(* Timer activ *)
	TimerOn(IN:=TRUE,PT:=T_Cylinder.T_Config.tDelayOn);
	TimerOff(IN:=TRUE,PT:=T_Cylinder.T_Config.tDelayOff);
	TimerPreOn(IN:=TRUE,PT:=T_Cylinder.T_Config.tDelayPreOn);
	TimerPreOff(IN:=TRUE,PT:=T_Cylinder.T_Config.tDelayPreOff);
	TimerOut(IN:=TRUE,PT:=T_Cylinder.T_Config.tTimeOut);
	TimerActiv(IN:=TRUE,PT:=T_Cylinder.T_CtrleCyl.T_Standard.tDelayActiv);
	TimerAfterSensorOn(IN:=TRUE,PT:=T_Cylinder.T_CtrleCyl.T_Standard.tDelayAfterSensorOn);
	TimerAfterSensorOff(IN:=TRUE,PT:=T_Cylinder.T_CtrleCyl.T_Standard.tDelayAfterSensorOff);
(* waiting for activ *)
	IF NOT(T_Cylinder.T_CtrleCyl.xErr) THEN
		CASE iStep OF
		(* process timer On *)
		1:	IF (T_Cylinder.T_Config.tDelayPreOn = T#0s) THEN
				TimerOn(IN:=FALSE);
				xCylinder:=T_Cylinder.T_Config.xActivState;
				T_Cylinder.T_CtrleCyl.T_Standard.xActivOn:=TRUE;
				iStep:=2;
			ELSE
				TimerPreOn(IN:=FALSE);
				iStep:=4;
			END_IF;
		(* wait for timer On *)
		2:	IF TimerOn.Q THEN
				iStep:=3;
				TimerOut(IN:=FALSE);
			END_IF
		(* control position activ *)
		3:	IF T_Cylinder.T_Config.xCtrlePosOn THEN
			(* position ctrle activ *)
				IF TimerOut.Q THEN
				(* timerout done, activ error cylinder has not activ position reached *)
					iStep:=999;
				ELSE
					IF xCtrlePosOn THEN
					(* Activ position reached, activ confirmation *)
						iStep:=80;
					END_IF
				END_IF
			ELSE
			(* no position ctrle, activ confirm *)
				iStep:=90;
			END_IF
		(* wait for timer Pre On *)
		4:	IF TimerPreOn.Q THEN
				T_Cylinder.T_Config.tDelayPreOn:=T#0s;
				iStep:=1;
			END_IF
		(* process timer Off *)
		11:	IF (T_Cylinder.T_Config.tDelayPreOff = T#0s) THEN
				TimerOff(IN:=FALSE);
				xCylinder:=NOT(T_Cylinder.T_Config.xActivState);
				T_Cylinder.T_CtrleCyl.T_Standard.xActivOn:=FALSE;
				iStep:=12;
			ELSE
				TimerPreOff(IN:=FALSE);
				iStep:=14;
			END_IF;
		(* wait for timer Off *)
		12:	IF TimerOff.Q THEN
				iStep:=13;
				TimerOut(IN:=FALSE);
			END_IF
		(* control position inactiv *)
		13:	IF T_Cylinder.T_Config.xCtrlePosOff THEN
			(* control position activ *)
				IF TimerOut.Q THEN
				(* timerout done, activ error 'cylinder has not inactiv position reached' *)
					iStep:=998;
				ELSE
					IF xCtrlePosOff THEN
					(* inactiv position reached, activ confirmation *)
						iStep:=85;
					END_IF
				END_IF
			ELSE
			(* no control position activ, activ confirmation *)
				iStep:=99;
			END_IF
		(* wait for timer Pre Off *)
		14:	IF TimerPreOff.Q THEN
				T_Cylinder.T_Config.tDelayPreOff:=T#0s;
				iStep:=11;
			END_IF
		(* inverse cylinder state *)
		51:	xCylinder:=NOT(xCylinder);
			T_Cylinder.T_CtrleCyl.T_Standard.xActivOn:=NOT(T_Cylinder.T_CtrleCyl.T_Standard.xActivOn);
			iStep:=99;
		80:	IF (T_Cylinder.T_CtrleCyl.T_Standard.tDelayAfterSensorOn <> T#0s) THEN
				TimerAfterSensorOn(IN:=FALSE);
				iStep:=81;
			ELSE
				iStep:=90;
			END_IF;
		(* wait for time after sensor *)
		81:	IF TimerAfterSensorOn.Q THEN
				iStep:=90;
			END_IF
		85:	IF (T_Cylinder.T_CtrleCyl.T_Standard.tDelayAfterSensorOff <> T#0s) THEN
				TimerAfterSensorOff(IN:=FALSE);
				iStep:=86;
			ELSE
				iStep:=99;
			END_IF;
		(* wait for time after sensor *)
		86:	IF TimerAfterSensorOff.Q THEN
				iStep:=99;
			END_IF
		(* test if delay activ *)
		90:	IF T_Cylinder.T_CtrleCyl.T_Standard.tDelayActiv <> T#0s THEN
				TimerActiv(IN:=FALSE);
				iStep:=98;
			ELSE
				iStep:=99;
			END_IF
		(* wait for time delay activ *)
		98:	IF TimerActiv.Q THEN
			(* activ time is over, set variable off *)
				xCylinder:=NOT(T_Cylinder.T_Config.xActivState);
				T_Cylinder.T_CtrleCyl.T_Standard.xActivOn:=FALSE;
				iStep:=99;
			END_IF
		(* process end *)
		99:	T_Cylinder.T_CtrleCyl.xDone:=TRUE;
			T_Cylinder.T_CtrleCyl.xErr:=FALSE;
			T_Cylinder.T_CtrleCyl.udiErrorID:=16#0;
		(* error, cylinder not in inactiv position *)
		998:	T_Cylinder.T_CtrleCyl.xDone:=FALSE;
			T_Cylinder.T_CtrleCyl.xErr:=TRUE;
			T_Cylinder.T_CtrleCyl.udiErrorID:=16#F202;
		(* error, cylinder not in activ position *)
		999:	T_Cylinder.T_CtrleCyl.xDone:=FALSE;
			T_Cylinder.T_CtrleCyl.xErr:=TRUE;
			T_Cylinder.T_CtrleCyl.udiErrorID:=16#F201;
		END_CASE
	END_IF;
END_FUNCTION_BLOCK

(* POU GENERAL/FB_CalcSpindleForce, ST *)
FUNCTION_BLOCK FB_CalcSpindleForce
VAR_INPUT
	rForcePistonIn:REAL;	(* in Newton *)
	rPistonDiameterD1:REAL;	(* in mm *)
	rPistonDiameterD2:REAL;	(* in mm *)
	rMaxAirpressure:REAL;		(* in bar *)
	rMaxServoVoltage:REAL;	(* in Volt *)
END_VAR
VAR_OUTPUT
	iAnalogOutput:INT;		(* range 0 - 32767 *)
	rSetMaxForce:REAL;		(* in Newton *)
	rForcePistonOut:REAL;	(* in Newton *)
END_VAR
VAR
	rMaxForce: REAL;
	rAreaOutside: REAL;
	rArea: REAL;
	rTmpMaxAirpressure: REAL;
	rTmpAnalogOut:REAL;
	rMaxDigitAnalogOutput: REAL;
END_VAR
	rMaxDigitAnalogOutput:=(32767.0 / 10.0) * rMaxServoVoltage;
	rAreaOutside:=((rPistonDiameterD1/2.0)*(rPistonDiameterD1/2.0))*PI;
	rArea:=ABS(rAreaOutside) * 2.0;	(* the new spindle has two piston *)
	rArea:=rArea / 1000000.0;	(* Umwandeln von mm^2 in m^2 *)
	rTmpMaxAirpressure:=rMaxAirpressure * 100000.0;	(* convert from bar to pascal *)
	rMaxForce:=rArea * rTmpMaxAirpressure;
	rSetMaxForce:=rMaxForce;
	IF(rMaxForce = 0) THEN rMaxForce:=0.01; END_IF;	(* check divide by zero *)
	IF(rMaxForce <> 0.0) THEN
		rTmpAnalogOut:=(rForcePistonIn/rMaxForce)*rMaxDigitAnalogOutput;
		IF (rTmpAnalogOut > rMaxDigitAnalogOutput) THEN
			iAnalogOutput:=REAL_TO_INT(rMaxDigitAnalogOutput);
		ELSE
			iAnalogOutput:=REAL_TO_INT(rTmpAnalogOut);
		END_IF;
		rForcePistonOut:=rForcePistonIn;
	ELSE
		iAnalogOutput:=0;
		rForcePistonOut:=0;
	END_IF;
END_FUNCTION_BLOCK

(* POU GENERAL/FB_TorqueLevelAirPressureAnalog, ST *)
FUNCTION_BLOCK FB_TorqueLevelAirPressureAnalog
VAR_INPUT
	xActiveWorkProcess:BOOL;
	xBlockOutput:BOOL;
	rForceIn:REAL;			(* Range 0 - MaxTorque (mNm) *)
	T_Station_Parameter:ST_RETAIN_DATA_STATIONWORK;
	lrZ1ActualPosition:LREAL;
	xCylHCActive:BOOL;
END_VAR
VAR_OUTPUT
	iAnalogOutput:INT;		(* Range 0 - 32767 *)
	rForceOut:REAL;			(* Range 0 - MaxTorque (mNm) *)
	rMaxTorque:REAL;		(* mNm *)
END_VAR
VAR_IN_OUT
	TCylTorque:ST_CYLINDER;
END_VAR
VAR
	rTorque:REAL;
	rTorqueEndPosition:REAL;
	rAirPressureP:REAL;
	rDiffTorqueLEvel:REAL;
(* Tmp variable *)
	rMaxAirPressure: REAL;
	rTmpAnalogOut:REAL;
	rTmpForceOut: REAL;
	rPistonArea: REAL;
	rGearRatioGearBox: REAL;
	rPlanetCarrier: REAL;
	rGearRatioRocker: REAL;
	rMaxTmpAirPressure: REAL;
	rTorqueStartPosition: REAL;
	rZ1Position: REAL;
	rZ1Length: REAL;
	rTorqueLevel1_StartPosition: REAL;
	rTorqueLevel1_EndPosition: REAL;
	rMaxDigitAnalogOutput: REAL;
END_VAR
IF xCylHCActive THEN
	rMaxDigitAnalogOutput:=(32767.0 / 10.0) * T_Station_Parameter.T_TorqueSystem.rMaxServoVoltage_HC;
	rPistonArea:=((T_Station_Parameter.T_TorqueSystem.rPistonTorqueHC/2.0)*(T_Station_Parameter.T_TorqueSystem.rPistonTorqueHC/2.0)*PI)/1000000.0;	(* Umwandlung in Quadratmeter *)
	rMaxAirPressure:=T_Station_Parameter.T_TorqueSystem.rMaxServoAirPressure_HC;
ELSE
	rMaxDigitAnalogOutput:=(32767.0 / 10.0) * T_Station_Parameter.T_TorqueSystem.rMaxServoVoltage_HCOver;
	rPistonArea:=((T_Station_Parameter.T_TorqueSystem.rPistonTorqueHCOverload/2.0)*(T_Station_Parameter.T_TorqueSystem.rPistonTorqueHCOverload/2.0)*PI)/1000000.0;	(* Umwandlung in Quadratmeter *)
	rMaxAirPressure:=T_Station_Parameter.T_TorqueSystem.rMaxServoAirPressure_HCOver;
END_IF;
rGearRatioGearBox:=T_Station_Parameter.T_TorqueSystem.rGearRatioGearBox;
rGearRatioRocker:=T_Station_Parameter.T_TorqueSystem.rGearRatioRocker;
rPlanetCarrier:=T_Station_Parameter.T_TorqueSystem.rPlanetCarrier_Radius;
rTorque:=rForceIn;		(* in mNm *)
rTorqueLevel1_StartPosition:=T_Station_Parameter.T_OnlineChange.rTorqueLevelHC;
rTorqueLevel1_EndPosition:=T_Station_Parameter.T_OnlineChange.rTorqueLevelHC;
IF ((rPlanetCarrier * rPistonArea) <> 0.0) AND (rMaxAirPressure <> 0.0) AND ((1.0 - rGearRatioGearBox) <> 0.0) THEN
	rAirPressureP:=(rTorque - (rTorque * rGearRatioGearBox))/(rPlanetCarrier * rPistonArea);	(* Pascal *)
	rAirPressureP:=rAirPressureP / 100000.0;	(* convert in bar *)
	rTmpAnalogOut:=((rMaxDigitAnalogOutput/rMaxAirPressure)*rAirPressureP);
	rMaxTmpAirPressure:=rMaxAirPressure * 100000.0;		(* convert from bar to pascal *)
	rMaxTorque:=(rMaxTmpAirPressure * rPlanetCarrier * rPistonArea) / (1.0 - rGearRatioGearBox);
	rMaxTorque:=(rMaxTorque / 32767.0) * rMaxDigitAnalogOutput;
ELSE
	rAirPressureP:=0.0;
	rMaxTmpAirPressure:=0.0;
	rMaxTorque:=0.0;
END_IF;
IF xActiveWorkProcess THEN
	(* Drehmoment wird in Abhängigkeit der Z1 Achse Position gesetzt *)
	rTorqueStartPosition:=(rTorqueLevel1_StartPosition + T_Station_Parameter.T_Fct_SpindleCalibration.arOffsetToolTorque[1]);
	rTorqueEndPosition:=(rTorqueLevel1_EndPosition + T_Station_Parameter.T_Fct_SpindleCalibration.arOffsetToolTorque[1]);
	IF ((rPlanetCarrier * rPistonArea) <> 0.0) AND (rMaxAirPressure <> 0.0) AND ((1.0 - rGearRatioGearBox) <> 0.0) THEN
		IF NOT(xBlockOutput) THEN
			IF (lrZ1ActualPosition >= grZ_WorkStartPos) THEN
				rZ1Length:=ABS(grZ_WorkStartPos - garPositionEndProcCalc[1]);
				rZ1Position:=ABS(lrZ1ActualPosition - grZ_WorkStartPos);
				rDiffTorqueLevel:=rTorqueEndPosition - rTorqueStartPosition;
				IF (rZ1Length <> 0.0) THEN
					rTorque:=rTorqueStartPosition + ((rDiffTorqueLevel / rZ1Length) * rZ1Position);
					rAirPressureP:=(rTorque - (rTorque * rGearRatioGearBox))/(rPlanetCarrier * rPistonArea);	(* Pascal *)
					rAirPressureP:=rAirPressureP / 100000.0;	(* convert in bar *)
					rTmpAnalogOut:=((rMaxDigitAnalogOutput/rMaxAirPressure)*rAirPressureP);
					rTmpForceOut:=rTorque;
				ELSE
					rTmpAnalogOut:=0.0;
					rTmpForceOut:=0.0;
				END_IF;
				IF NOT(TCylTorque.T_CtrleCyl.xExecute) AND TCylTorque.T_CtrleCyl.xDone THEN
					TCylTorque.T_CtrleCyl.iFunction:=4;
					TCylTorque.T_CtrleCyl.xExecute:=TRUE;
				END_IF;
			END_IF
		END_IF;
	END_IF;
ELSE
	rTmpForceOut:=rForceIn;
END_IF;
(* Set Output value *)
rForceOut:=rTmpForceOut;
IF (rTmpAnalogOut < 32767.0) AND (rTmpAnalogOut >= 0.0) THEN
	iAnalogOutput:=REAL_TO_INT(rTmpAnalogOut);
ELSIF (rTmpAnalogOut >= 32767.0) THEN
	iAnalogOutput:=32767;
ELSIF (rTmpAnalogOut < 0.0) THEN
	iAnalogOutput:=0;
END_IF;
END_FUNCTION_BLOCK

(* POU FB_HARDWARE/FBHW_CYL_STANDARD_2WAY, ST *)
FUNCTION_BLOCK FBHW_CYL_STANDARD_2WAY
VAR_INPUT
	xCtrlePosOn:BOOL;
	xCtrlePosOff:BOOL;
END_VAR
VAR_OUTPUT
	xCylinderOn:BOOL;
	xCylinderOff:BOOL;
END_VAR
VAR_IN_OUT
	T_Cylinder:ST_CYLINDER;
END_VAR
VAR
(* variable *)
	xConfirmResetFB:BOOL:=FALSE;
	iStep:INT;
(* timer *)
	TimerOn:TON;
	TimerOff:TON;
	TimerPreOn:TON;
	TimerPreOff:TON;
	TimerOut:TON;
	TimerActiv: TON;
(* trigger *)
	RisingEdgeActiv:R_TRIG;
	FallingEdgeActiv:F_TRIG;
	RisingEdgeReset:R_TRIG;
	RisingEdgeExecute:R_TRIG;
	TimerAfterSensorOn: TON;
	TimerAfterSensorOff: TON;
	TONWaitSwitch: TON;
END_VAR
(* if function bloc set activ then Analog state will be transfered *)
	RisingEdgeActiv(CLK:=T_Cylinder.T_CtrleCyl.xFBActiv);
	FallingEdgeActiv(CLK:=T_Cylinder.T_CtrleCyl.xFBActiv);
	IF RisingEdgeActiv.Q OR FallingEdgeActiv.Q THEN
	(* set Analog Out = In on the rising edge from the activ signal *)
		xCylinderOn:=NOT(T_Cylinder.T_Config.xActivState);
		xCylinderOff:=NOT(T_Cylinder.T_Config.xActivState);
		T_Cylinder.T_CtrleCyl.T_Standard.xActivOn:= FALSE;
		T_Cylinder.T_CtrleCyl.T_Standard.xActivOff:= FALSE;
	END_IF

(* if bloc disable if activ signal is inactiv *)
	IF T_Cylinder.T_CtrleCyl.xFBActiv THEN
	(* copy control position state *)
		T_Cylinder.T_CtrleCyl.xStatePosOn:=xCtrlePosOn;
		T_Cylinder.T_CtrleCyl.xStatePosOff:=xCtrlePosOff;
	ELSE
	(* exit FB *)
		RETURN;
	END_IF

(* wait for reseting *)
	RisingEdgeReset(CLK:=T_Cylinder.T_CtrleCyl.xReset);
	IF RisingEdgeReset.Q THEN
		(* Init. timer *)
		TimerOn(IN:=TRUE,PT:=T#1ms);
		TimerOff(IN:=TRUE,PT:=T#1ms);
		TimerPreOn(IN:=TRUE,PT:=T#1ms);
		TimerPreOff(IN:=TRUE,PT:=T#1ms);
		TimerOut(IN:=TRUE,PT:=T#1ms);
	(* Init. variable *)
		iStep:=0;
	(* Init. structure *)
		T_Cylinder.T_CtrleCyl.iFunction:=0;
		T_Cylinder.T_CtrleCyl.T_Standard.xActivOn:= FALSE;
		T_Cylinder.T_CtrleCyl.T_Standard.xActivOff:= FALSE;
		xCylinderOn:=NOT(T_Cylinder.T_Config.xActivState);
		xCylinderOff:=NOT(T_Cylinder.T_Config.xActivState);
		T_Cylinder.T_CtrleCyl.xDone:=FALSE;
		T_Cylinder.T_CtrleCyl.xErr:=FALSE;
		T_Cylinder.T_CtrleCyl.udiErrorID:=16#0;
	(* confirm reset *)
		xConfirmResetFB:=TRUE;
	(* exit function *)
		RETURN;
	ELSE
		IF xConfirmResetFB THEN
		(* confirm reset FB *)
			T_Cylinder.T_CtrleCyl.xDone:=TRUE;
			T_Cylinder.T_CtrleCyl.xErr:=FALSE;
			T_Cylinder.T_CtrleCyl.udiErrorID:=16#0;
			(* reset variable *)
			xConfirmResetFB:=FALSE;
		END_IF
	END_IF

(* if bloc disable if activ signal is inactiv *)
	IF NOT(T_Cylinder.T_CtrleCyl.xFBActiv) THEN
		RETURN;
	END_IF

(* wait for execute *)
	RisingEdgeExecute(CLK:=T_Cylinder.T_CtrleCyl.xExecute);
	IF RisingEdgeExecute.Q THEN
		IF NOT(T_Cylinder.T_CtrleCyl.xDone) AND NOT(T_Cylinder.T_CtrleCyl.xErr) THEN
		(* can execute function if both signal are disable *)
			RETURN;
		END_IF
		CASE T_Cylinder.T_CtrleCyl.iFunction OF
		(* disable *)
		1:	iStep:=11;
		(* Activ without sensor position ctrle *)
		2:	iStep:=1;
		(* inverse cylinder state *)
		51:	iStep:=51;
		ELSE
			(* function not implemented *)
			iStep:=0;
			T_Cylinder.T_CtrleCyl.xDone:=FALSE;
			T_Cylinder.T_CtrleCyl.xErr:=TRUE;
			T_Cylinder.T_CtrleCyl.udiErrorID:=16#F000;
			(* exit FB *)
			RETURN;
		END_CASE
		(* Init. variable *)
		T_Cylinder.T_CtrleCyl.xDone:=FALSE;
		T_Cylinder.T_CtrleCyl.xErr:=FALSE;
		T_Cylinder.T_CtrleCyl.udiErrorID:=16#0;
		(* exit FB *)
		RETURN;
	END_IF

(* Timer activ *)
	TimerOn(IN:=TRUE,PT:=T_Cylinder.T_Config.tDelayOn);
	TimerOff(IN:=TRUE,PT:=T_Cylinder.T_Config.tDelayOff);
	TimerPreOn(IN:=TRUE,PT:=T_Cylinder.T_Config.tDelayPreOn);
	TimerPreOff(IN:=TRUE,PT:=T_Cylinder.T_Config.tDelayPreOff);
	TimerOut(IN:=TRUE,PT:=T_Cylinder.T_Config.tTimeOut);
	TimerActiv(IN:=TRUE,PT:=T_Cylinder.T_CtrleCyl.T_Standard.tDelayActiv);
	TimerAfterSensorOn(IN:=TRUE,PT:=T_Cylinder.T_CtrleCyl.T_Standard.tDelayAfterSensorOn);
	TimerAfterSensorOff(IN:=TRUE,PT:=T_Cylinder.T_CtrleCyl.T_Standard.tDelayAfterSensorOff);

(* waiting for activ *)
	IF NOT(T_Cylinder.T_CtrleCyl.xErr) THEN
		CASE iStep OF
		(* process timer On *)
		1:	IF NOT(xCylinderOn) AND NOT(xCylinderOff) THEN
				iStep:=5;
				xCylinderOn:=FALSE;
				xCylinderOff:=TRUE;
				TONWaitSwitch(IN:=FALSE);
				RETURN;
			END_IF;
			IF (T_Cylinder.T_Config.tDelayPreOn = T#0s) THEN
				TimerOn(IN:=FALSE);
				xCylinderOn:=T_Cylinder.T_Config.xActivState;
				xCylinderOff:=NOT(T_Cylinder.T_Config.xActivState);
				T_Cylinder.T_CtrleCyl.T_Standard.xActivOn:= TRUE;
				T_Cylinder.T_CtrleCyl.T_Standard.xActivOff:= FALSE;
				iStep:=2;
			ELSE
				TimerPreOn(IN:=FALSE);
				iStep:=4;
			END_IF;
		(* wait for timer On *)
		2:	IF TimerOn.Q THEN
				iStep:=3;
				TimerOut(IN:=FALSE);
			END_IF
		(* control position activ *)
		3:	IF T_Cylinder.T_Config.xCtrlePosOn THEN
			(* position ctrle activ *)
				IF TimerOut.Q THEN
				(* timerout done, activ error cylinder has not activ position reached *)
					iStep:=999;
				ELSE
					IF xCtrlePosOn THEN
					(* Activ position reached, activ confirmation *)
						iStep:=80;
					END_IF
				END_IF
			ELSE
			(* no position ctrle, activ confirm *)
				iStep:=90;
			END_IF
		(* wait for timer Pre On *)
		4:	IF TimerPreOn.Q THEN
				T_Cylinder.T_Config.tDelayPreOn:=T#0s;
				iStep:=1;
			END_IF
		5:	TONWaitSwitch(IN:=TRUE,PT:=T#0.1s);
			IF TONWaitSwitch.Q THEN
				TONWaitSwitch(IN:=FALSE);
				iStep:=1;
			END_IF;
		(* process timer Off *)
		11:	IF NOT(xCylinderOn) AND NOT(xCylinderOff) THEN
				iStep:=15;
				xCylinderOn:=FALSE;
				xCylinderOff:=TRUE;
				TONWaitSwitch(IN:=FALSE);
				RETURN;
			END_IF;
			IF (T_Cylinder.T_Config.tDelayPreOff = T#0s) THEN
				TimerOff(IN:=FALSE);
				xCylinderOn:=NOT(T_Cylinder.T_Config.xActivState);
				xCylinderOff:=T_Cylinder.T_Config.xActivState;
				T_Cylinder.T_CtrleCyl.T_Standard.xActivOn:= FALSE;
				T_Cylinder.T_CtrleCyl.T_Standard.xActivOff:= TRUE;
				iStep:=12;
			ELSE
				TimerPreOff(IN:=FALSE);
				iStep:=14;
			END_IF;
		(* wait for timer Off *)
		12:	IF TimerOff.Q THEN
				iStep:=13;
				TimerOut(IN:=FALSE);
			END_IF
		(* control position inactiv *)
		13:	IF T_Cylinder.T_Config.xCtrlePosOff THEN
			(* control position activ *)
				IF TimerOut.Q THEN
				(* timerout done, activ error 'cylinder has not inactiv position reached' *)
					iStep:=998;
				ELSE
					IF xCtrlePosOff THEN
					(* inactiv position reached, activ confirmation *)
						iStep:=85;
					END_IF
				END_IF
			ELSE
			(* no control position activ, activ confirmation *)
				iStep:=99;
			END_IF
		(* wait for timer Pre Off *)
		14:	IF TimerPreOff.Q THEN
				T_Cylinder.T_Config.tDelayPreOff:=T#0s;
				iStep:=11;
			END_IF
		15:	TONWaitSwitch(IN:=TRUE,PT:=T#0.1s);
			IF TONWaitSwitch.Q THEN
				TONWaitSwitch(IN:=FALSE);
				iStep:=11;
			END_IF;
		(* inverse cylinder state *)
		51:	IF xCylinderOn THEN
				xCylinderOn:=FALSE;
				xCylinderOff:=TRUE;
				T_Cylinder.T_CtrleCyl.T_Standard.xActivOn:=FALSE;
				T_Cylinder.T_CtrleCyl.T_Standard.xActivOff:=TRUE;
				iStep:=99;
			ELSIF xCylinderOff THEN
				xCylinderOff:=FALSE;
				xCylinderOn:=TRUE;
				T_Cylinder.T_CtrleCyl.T_Standard.xActivOn:=TRUE;
				T_Cylinder.T_CtrleCyl.T_Standard.xActivOff:=FALSE;
				iStep:=99;
			ELSE
				xCylinderOn:=FALSE;
				xCylinderOff:=FALSE;
				TONWaitSwitch(IN:=FALSE);
				iStep:=52;
			END_IF;
		52:	TONWaitSwitch(IN:=TRUE,PT:=T#0.1s);
			IF TONWaitSwitch.Q THEN
				TONWaitSwitch(IN:=FALSE);
				xCylinderOn:=FALSE;
				xCylinderOff:=TRUE;
				T_Cylinder.T_CtrleCyl.T_Standard.xActivOn:=FALSE;
				T_Cylinder.T_CtrleCyl.T_Standard.xActivOff:=TRUE;
				iStep:=99;
			END_IF;
		80:	IF (T_Cylinder.T_CtrleCyl.T_Standard.tDelayAfterSensorOn <> T#0s) THEN
				TimerAfterSensorOn(IN:=FALSE);
				iStep:=81;
			ELSE
				iStep:=90;
			END_IF;
		(* wait for time after sensor *)
		81:	IF TimerAfterSensorOn.Q THEN
				iStep:=90;
			END_IF
		85:	IF (T_Cylinder.T_CtrleCyl.T_Standard.tDelayAfterSensorOff <> T#0s) THEN
				TimerAfterSensorOff(IN:=FALSE);
				iStep:=86;
			ELSE
				iStep:=99;
			END_IF;
		(* wait for time after sensor *)
		86:	IF TimerAfterSensorOff.Q THEN
				iStep:=99;
			END_IF
		(* test if delay activ *)
		90:	IF T_Cylinder.T_CtrleCyl.T_Standard.tDelayActiv <> T#0s THEN
				TimerActiv(IN:=FALSE);
				iStep:=98;
			ELSE
				iStep:=99;
			END_IF
		(* wait for time delay activ *)
		98:	IF TimerActiv.Q THEN
			(* activ time is over, set variable off *)
				xCylinderOn:=NOT(T_Cylinder.T_Config.xActivState);
				xCylinderOff:=NOT(T_Cylinder.T_Config.xActivState);
				T_Cylinder.T_CtrleCyl.T_Standard.xActivOn:=FALSE;
				T_Cylinder.T_CtrleCyl.T_Standard.xActivOff:=FALSE;
				iStep:=99;
			END_IF
		(* process end *)
		99:	T_Cylinder.T_CtrleCyl.xDone:=TRUE;
			T_Cylinder.T_CtrleCyl.xErr:=FALSE;
			T_Cylinder.T_CtrleCyl.udiErrorID:=16#0;
		(* error, cylinder not in inactiv position *)
		998:	T_Cylinder.T_CtrleCyl.xDone:=FALSE;
			T_Cylinder.T_CtrleCyl.xErr:=TRUE;
			T_Cylinder.T_CtrleCyl.udiErrorID:=16#F202;
		(* error, cylinder not in activ position *)
		999:	T_Cylinder.T_CtrleCyl.xDone:=FALSE;
			T_Cylinder.T_CtrleCyl.xErr:=TRUE;
			T_Cylinder.T_CtrleCyl.udiErrorID:=16#F201;
		END_CASE
	END_IF;
END_FUNCTION_BLOCK

(* POU FB_HARDWARE/FB_ReadAxisState, ST *)
FUNCTION_BLOCK FB_ReadAxisState
VAR_INPUT
	bExecute			:BOOL;
	iFunctionNr			:INT;
	nSlaveAddr			:INT;
	nSubIndex			:BYTE;
END_VAR
VAR_IN_OUT
	T_AxisRefIn:NCTOPLC_AXLESTRUCT;
END_VAR
VAR_OUTPUT
	Done				:BOOL;		(* successfully done *)
	dwValueOut: DWORD;
END_VAR
VAR
	fbCoEReadParameter 		: FB_EcCoESdoRead;
	abyReceive				: ARRAY[0..10] OF BYTE;
	state					:INT;
	Trigger					:R_TRIG;
	fbGetAmsNetID			 : FB_GetAxisAmsAddr;
	sEtherCATNetId 			: STRING;	(*Master Ethercat AMS Adress *)
END_VAR
Trigger( CLK:=bExecute );
IF Trigger.Q THEN
	CASE iFunctionNr OF
		(* Lesen der NetID und abfragen des Status füs Achse Safety Funktionen *)
		1:	state:=1;
	END_CASE;
	Done := FALSE;
END_IF;
CASE state OF
(*		get AMS Net ID of the Drive-Unit*)
(*************************************************************************************************************************)
	1:	fbGetAmsNetID(	sNetId:= '',
						iAxisId:= DWORD_TO_UINT(T_AxisRefIn.nAxisId),
						bExecute := TRUE);
		IF NOT fbGetAmsNetID.bBusy AND NOT fbGetAmsNetID.bError THEN
			fbGetAmsNetID.AxisNetId;
			sEtherCATNetId 	:= fbGetAmsNetID.AxisNetId;
			fbGetAmsNetID(	sNetId:= '',
							iAxisId:= DWORD_TO_UINT(T_AxisRefIn.nAxisId),
							bExecute := FALSE);
			state := 10;
		END_IF
(*************************************************************************************************************************)
	10:	fbCoEReadParameter.nIndex		:= 16#FA10;
		fbCoEReadParameter.nSubIndex	:=nSubIndex;
		fbCoEReadParameter.cbBufLen		:=2;
		fbCoEReadParameter.bExecute 	:= TRUE;
		state := 11;
	11: 	IF NOT fbCoEReadParameter.bBusy THEN
			fbCoEReadParameter.bExecute 	:= FALSE;
			state := 0;
			Done := TRUE;
			dwValueOut:=abyReceive[0] + (abyReceive[1] * 256);
		END_IF;
(*************************************************************************************************************************)
 END_CASE
fbCoEReadParameter(		sNetId		:= sEtherCATNetId,
						nSlaveAddr	:= nSlaveAddr,
						tTimeout		:= T#500ms,
						pDstBuf		:=ADR(abyReceive));
END_FUNCTION_BLOCK

(* POU FB_HARDWARE/FB_WriteObject, ST *)
FUNCTION_BLOCK FB_WriteObject
VAR_INPUT
	bExecute			:BOOL;
	iFunctionNr			:INT;
	nSlaveAddr			:INT;
	T_RegulatorSpindle:ST_EXCHG_PARAM_CONTRMOT;
END_VAR
VAR_IN_OUT
	T_AxisRefIn:NCTOPLC_AXLESTRUCT;
END_VAR
VAR_OUTPUT
	Done				:BOOL;		(* successfully done *)
	dwValueOut: DWORD;
END_VAR
VAR
	fbCoEWriteParameter 		: FB_EcCoESdoWrite;
	abyReceive				: ARRAY[0..10] OF BYTE;
	state					:INT;
	Trigger					:R_TRIG;
	fbGetAmsNetID			 : FB_GetAxisAmsAddr;
	sEtherCATNetId 			: STRING;	(*Master Ethercat AMS Adress *)
	ii: INT;
END_VAR
Trigger( CLK:=bExecute );
IF Trigger.Q THEN
	CASE iFunctionNr OF
		(* Lesen der NetID und abfragen des Status füs Achse Safety Funktionen *)
		1:	state:=1;
	END_CASE;
	Done := FALSE;
END_IF;
CASE state OF
(*		get AMS Net ID of the Drive-Unit*)
(*************************************************************************************************************************)
	1:	fbGetAmsNetID(	sNetId:= '',
						iAxisId:= DWORD_TO_UINT(T_AxisRefIn.nAxisId),
						bExecute := TRUE);
		IF NOT fbGetAmsNetID.bBusy AND NOT fbGetAmsNetID.bError THEN
			fbGetAmsNetID.AxisNetId;
			sEtherCATNetId 	:= fbGetAmsNetID.AxisNetId;
			fbGetAmsNetID(	sNetId:= '',
							iAxisId:= DWORD_TO_UINT(T_AxisRefIn.nAxisId),
							bExecute := FALSE);
			FOR ii:=0 TO 10 DO
				abyReceive[ii]:=0;
			END_FOR;
			state := 10;
		END_IF
(*************************************************************************************************************************)
	10:	fbCoEWriteParameter(bExecute 	:= FALSE);
		fbCoEWriteParameter.nIndex		:= 16#60F6;	(* Current Control Parameter Set *)
		fbCoEWriteParameter.nSubIndex	:=1;
		dwValueOut:=abyReceive[0]:=INT_TO_BYTE(T_RegulatorSpindle.iCurrentReg_PGain);
		dwValueOut:=abyReceive[1]:=INT_TO_BYTE(T_RegulatorSpindle.iCurrentReg_PGain / 256);
		fbCoEWriteParameter.pSrcBuf		:=ADR(abyReceive);
		fbCoEWriteParameter.cbBufLen		:=SIZEOF(abyReceive);
		fbCoEWriteParameter.bExecute 	:= TRUE;
		state := 11;
	11: 	IF NOT fbCoEWriteParameter.bBusy THEN
			fbCoEWriteParameter(bExecute 	:= FALSE);
			fbCoEWriteParameter.nIndex		:= 16#60F6;	(* Current Control Parameter Set *)
			fbCoEWriteParameter.nSubIndex	:=2;
			dwValueOut:=abyReceive[0]:=INT_TO_BYTE(T_RegulatorSpindle.iCurrentReg_IGain);
			dwValueOut:=abyReceive[1]:=INT_TO_BYTE(T_RegulatorSpindle.iCurrentReg_IGain / 256);
			fbCoEWriteParameter.pSrcBuf		:=ADR(abyReceive);
			fbCoEWriteParameter.cbBufLen		:=SIZEOF(abyReceive);
			fbCoEWriteParameter.bExecute 	:= TRUE;
			state := 12;
		END_IF;
	12: 	IF NOT fbCoEWriteParameter.bBusy THEN
			fbCoEWriteParameter(bExecute 	:= FALSE);
			fbCoEWriteParameter.nIndex		:= 16#60F9;	(* Velocity Control Parameter Set *)
			fbCoEWriteParameter.nSubIndex	:=1;
			dwValueOut:=abyReceive[0]:=INT_TO_BYTE(T_RegulatorSpindle.iSpeedReg_PGain);
			dwValueOut:=abyReceive[1]:=INT_TO_BYTE(T_RegulatorSpindle.iSpeedReg_PGain / 256);
			fbCoEWriteParameter.pSrcBuf		:=ADR(abyReceive);
			fbCoEWriteParameter.cbBufLen		:=SIZEOF(abyReceive);
			fbCoEWriteParameter.bExecute 	:= TRUE;
			state := 13;
		END_IF;
	13: 	IF NOT fbCoEWriteParameter.bBusy THEN
			fbCoEWriteParameter(bExecute 	:= FALSE);
			fbCoEWriteParameter.nIndex		:= 16#60F9;	(* Velocity Control Parameter Set *)
			fbCoEWriteParameter.nSubIndex	:=2;
			dwValueOut:=abyReceive[0]:=INT_TO_BYTE(T_RegulatorSpindle.iSpeedReg_IGain);
			dwValueOut:=abyReceive[1]:=INT_TO_BYTE(T_RegulatorSpindle.iSpeedReg_IGain / 256);
			fbCoEWriteParameter.pSrcBuf		:=ADR(abyReceive);
			fbCoEWriteParameter.cbBufLen		:=SIZEOF(abyReceive);
			fbCoEWriteParameter.bExecute 	:= TRUE;
			state := 14;
		END_IF;
	14: 	IF NOT fbCoEWriteParameter.bBusy THEN
			fbCoEWriteParameter(bExecute 	:= FALSE);
			fbCoEWriteParameter.nIndex		:= 16#60FB;	(* Position Control Parameter Set *)
			fbCoEWriteParameter.nSubIndex	:=1;
			dwValueOut:=abyReceive[0]:=INT_TO_BYTE(T_RegulatorSpindle.iPositionReg_PGain);
			dwValueOut:=abyReceive[1]:=INT_TO_BYTE(T_RegulatorSpindle.iPositionReg_PGain / 256);
			fbCoEWriteParameter.pSrcBuf		:=ADR(abyReceive);
			fbCoEWriteParameter.cbBufLen		:=SIZEOF(abyReceive);
			fbCoEWriteParameter.bExecute 	:= TRUE;
			state := 15;
		END_IF;
	15: 	IF NOT fbCoEWriteParameter.bBusy THEN
			fbCoEWriteParameter(bExecute 	:= FALSE);
			fbCoEWriteParameter.nIndex		:= 16#60FB;	(* Position Control Parameter Set *)
			fbCoEWriteParameter.nSubIndex	:=2;
			dwValueOut:=abyReceive[0]:=INT_TO_BYTE(T_RegulatorSpindle.iPositionReg_IGain);
			dwValueOut:=abyReceive[1]:=INT_TO_BYTE(T_RegulatorSpindle.iPositionReg_IGain / 256);
			fbCoEWriteParameter.pSrcBuf		:=ADR(abyReceive);
			fbCoEWriteParameter.cbBufLen		:=SIZEOF(abyReceive);
			fbCoEWriteParameter.bExecute 	:= TRUE;
			state := 16;
		END_IF;
	16: 	IF NOT fbCoEWriteParameter.bBusy THEN
			fbCoEWriteParameter(bExecute 	:= FALSE);
			fbCoEWriteParameter.nIndex		:= 16#60FB;	(* Position Control Parameter Set *)
			fbCoEWriteParameter.nSubIndex	:=3;
			dwValueOut:=abyReceive[0]:=INT_TO_BYTE(T_RegulatorSpindle.iPositionReg_DGain);
			dwValueOut:=abyReceive[1]:=INT_TO_BYTE(T_RegulatorSpindle.iPositionReg_DGain / 256);
			fbCoEWriteParameter.pSrcBuf		:=ADR(abyReceive);
			fbCoEWriteParameter.cbBufLen		:=SIZEOF(abyReceive);
			fbCoEWriteParameter.bExecute 	:= TRUE;
			state := 17;
		END_IF;
	17: 	IF NOT fbCoEWriteParameter.bBusy THEN
			fbCoEWriteParameter(bExecute 	:= FALSE);
			fbCoEWriteParameter.nIndex		:= 16#2F10;	(* Store Parameter *)
			fbCoEWriteParameter.nSubIndex	:=1;
			dwValueOut:=abyReceive[0]:=16#73;	(* s *)
			dwValueOut:=abyReceive[1]:=16#61;	(* a *)
			dwValueOut:=abyReceive[2]:=16#76;	(* v *)
			dwValueOut:=abyReceive[3]:=16#65;	(* e *)
			fbCoEWriteParameter.pSrcBuf		:=ADR(abyReceive);
			fbCoEWriteParameter.cbBufLen		:=4;
			fbCoEWriteParameter.bExecute 	:= TRUE;
			state := 18;
		END_IF;
	18: 	IF NOT fbCoEWriteParameter.bBusy THEN
			fbCoEWriteParameter(bExecute 	:= FALSE);
			state := 0;
			Done := TRUE;
		END_IF;
(*************************************************************************************************************************)
 END_CASE
fbCoEWriteParameter(		sNetId		:= sEtherCATNetId,
						nSlaveAddr	:= nSlaveAddr,
						tTimeout		:= T#500ms);
END_FUNCTION_BLOCK

(* POU PRG_ERROR_WARNING_CTRLE, ST *)
PROGRAM PRG_ERROR_WARNING_CTRLE
VAR
	RisingEdge_ProcessError_St1St2: R_TRIG;
	RisingEdge_Station1Error: R_TRIG;
	RisingEdge_Station1_Axis1Error: R_TRIG;
	RisingEdge_Station1_Axis2Error: R_TRIG;
	RisingEdge_Station1_Axis3Error: R_TRIG;
	RisingEdge_Station2_Axis1Error: R_TRIG;
	RisingEdge_Station2_Axis2Error: R_TRIG;
	RisingEdge_Station2_Axis3Error: R_TRIG;
	RisingEdge_Station5_Axis1Error: R_TRIG;
	ii: INT;
	FBErrorMessage:FB_ErrorMessage;
	FBErrorMessageVisu:FB_ErrorMessage;
	diErrorNr: DINT;
	sErrorTimeStamp: STRING(12);
	RisingEdgeUpdateErrorList: R_TRIG;
	xNoProcessStationActive_St1St2: BOOL;
	iStepSetForceError: INT;
	adiTmpErrorList: ARRAY [1..20] OF DINT;
	asTmpErrorList: ARRAY [1..20] OF STRING(12);
	FBNT_GetTime:NT_GetTime;
	FBResetError: FB_ResetError;
	iStepResetError: INT;
	xSetError: BOOL;
	udi_TmpErrorNr: UDINT;
	TONWaitCheckError_Z_St1: TON;
	TONWaitCheckError_Z_St2: TON;
	TONWaitCheckError_S_St1: TON;
	TONWaitCheckError_S_St2: TON;
	TONWaitCheckError_O_St1: TON;
	TONWaitCheckError_O_St2: TON;
	TONWaitCheckError_C_St1: TON;
	xCheckAxisError_Z_St1: BOOL;
	xCheckAxisError_Z_St2: BOOL;
	xCheckAxisError_S_St1: BOOL;
	xCheckAxisError_S_St2: BOOL;
	xCheckAxisError_O_St1: BOOL;
	xCheckAxisError_O_St2: BOOL;
	xCheckAxisError_C_St1: BOOL;
	xExecuteResetError:BOOL;
END_VAR
IF (TStatusUPS.ePowerStatus = PowerOnBattery) THEN
	RETURN;
END_IF;
RisingEdge_ProcessError_St1St2(CLK:=NOT(TProcess.T_Ctrle.xDone) AND TProcess.T_Ctrle.xError);
RisingEdge_Station1Error(CLK:=NOT(TStation_Work_St1.TControl.xDone) AND TStation_Work_St1.TControl.xError);

RisingEdge_Station1_Axis1Error(CLK:=	NOT(TStation_Work_St1.THWWorkStation.TAxisZ.T_CtrleSingle.xDone) AND TStation_Work_St1.THWWorkStation.TAxisZ.T_CtrleSingle.xErr);
RisingEdge_Station1_Axis2Error(CLK:=	NOT(TStation_Work_St1.THWWorkStation.TAxisS.T_CtrleSingle.xDone) AND TStation_Work_St1.THWWorkStation.TAxisS.T_CtrleSingle.xErr);
IF RisingEdge_ProcessError_St1St2.Q AND T_StartUp.T_State.xCompleted THEN
	T_ExchgParam.T_SafetyCtrl.xSetForceError:=TRUE;
	T_ExchgParam.T_SafetyCtrl.diSetForceErrorNr:=TProcess.T_Ctrle.diErrorNr;
END_IF;
IF (TProcess.T_Ctrle.xDone AND NOT(TProcess.T_Ctrle.xError)) OR NOT(T_StartUp.T_State.xCompleted) THEN
	(* Stationsfehler nur auffangen falls der Prozess nicht aktiv ist oder die Maschine am Aufstarten ist *)
	IF RisingEdge_Station1Error.Q THEN
		T_ExchgParam.T_SafetyCtrl.xSetForceError:=TRUE;
		T_ExchgParam.T_SafetyCtrl.diSetForceErrorNr:=TStation_Work_St1.TControl.diErrorNr;
	END_IF;
END_IF;

AxisError;

IF (T_ExchgParam.T_SafetyCtrl.xSetForceError AND NOT(T_ExchgParam.T_SafetyCtrl.xResetErrorWarning)) OR xSetError THEN
	CASE iStepSetForceError OF
		1:	xSetError:=TRUE;
			T_VisuQVis.T_CtrleAction.xReset:=FALSE;
			T_StartUp.T_State.xBlockChangeMovementVisu:=FALSE;
			FBErrorMessage(	diErrorNr:=T_ExchgParam.T_SafetyCtrl.diSetForceErrorNr,
								T_ErrorList:=T_ErrorList);
			adiTmpErrorList:=T_NovRAM.T_Parameter.T_ErrorNrList.adiErrorListMachine;
			T_NovRAM.T_Parameter.T_ErrorNrList.adiErrorListMachine[1]:=T_ExchgParam.T_SafetyCtrl.diSetForceErrorNr;
			FOR ii:=2 TO 20 DO
				T_NovRAM.T_Parameter.T_ErrorNrList.adiErrorListMachine[ii]:=adiTmpErrorList[ii-1];
			END_FOR;
			iStepSetForceError:=iStepSetForceError + 1;
		2:	FBNT_GetTime(	NETID:= '',
							START:=FALSE );
			iStepSetForceError:=iStepSetForceError + 1;
		3:	FBNT_GetTime(	NETID:= '',
							START:= TRUE,
							TMOUT:= T#2s);
			IF NOT(FBNT_GetTime.BUSY) OR FBNT_GetTime.ERR THEN
				asTmpErrorList:=T_NovRAM.T_Parameter.T_ErrorNrList.asErrorTimeStampMachine;
				IF NOT(FBNT_GetTime.ERR) THEN
					T_NovRAM.T_Parameter.T_ErrorNrList.asErrorTimeStampMachine[1]:=Fct_ConvertDateToString(2,FBNT_GetTime.TIMESTR);
				ELSE
					T_NovRAM.T_Parameter.T_ErrorNrList.asErrorTimeStampMachine[1]:='00.00 00:00';	(* Fehler beim lesen der Systemzeit, daher wird ein default-Wert gesetzt *)
				END_IF;
				FOR ii:=2 TO 20 DO
					T_NovRAM.T_Parameter.T_ErrorNrList.asErrorTimeStampMachine[ii]:=asTmpErrorList[ii-1];
				END_FOR;
				iStepSetForceError:=iStepSetForceError + 1;
			END_IF;
		4:	IF NOT(T_VisuQVis.T_CtrleAction.xDone) AND NOT(T_VisuQVis.T_CtrleAction.xExecute) THEN
				T_VisuQVis.T_CtrleAction.xReset:=TRUE;
				iStepSetForceError:=iStepSetForceError + 1;
			END_IF;
			IF T_VisuQVis.T_CtrleAction.xDone AND NOT(T_VisuQVis.T_CtrleAction.xExecute) THEN
				iStepSetForceError:=iStepSetForceError + 1;
			END_IF;
		5:	IF T_VisuQVis.T_CtrleAction.xDone AND NOT(T_VisuQVis.T_CtrleAction.xReset) AND NOT(T_NovRAM.T_Ctrle.xExecute) AND T_NovRAM.T_Ctrle.xDone AND NOT(gxHardwareOFF) THEN
				T_NovRAM.T_Ctrle.xExecute:=TRUE;
				T_NovRAM.T_Ctrle.iFunction:=2;
				iStepSetForceError:=iStepSetForceError + 1;
			ELSE
				iStepSetForceError:=iStepSetForceError + 1;
			END_IF;
		6:	IF (NOT(T_NovRAM.T_Ctrle.xExecute) AND T_NovRAM.T_Ctrle.xDone) OR gxHardwareOFF THEN
				T_ExchgParam.T_SafetyCtrl.xUpdateErrorList:=TRUE;
				T_ExchgParam.T_Visu.T_Message.sDynamicTextEnglish:=FBErrorMessage.sErrorTextEnglish;
				T_ExchgParam.T_Visu.T_Message.sDynamicTextDeutsch:=FBErrorMessage.sErrorTextDeutsch;
				T_ExchgParam.T_Visu.T_Message.sDynamicTextFrancais:=FBErrorMessage.sErrorTextFrancais;
				iStepSetForceError:=iStepSetForceError + 1;
			END_IF;
		7:	IF (NOT(T_NovRAM.T_Ctrle.xExecute) AND T_NovRAM.T_Ctrle.xDone) OR gxHardwareOFF THEN
				iStepSetForceError:=1;
				T_ExchgParam.T_SafetyCtrl.xSetForceError:=FALSE;
				xSetError:=FALSE;
			END_IF;
	END_CASE;
ELSE
	iStepSetForceError:=1;
END_IF;

(* Monitor dynamic text *)
	IF (T_ExchgParam.T_Visu.T_Message.sDynamicTextEnglish <> '')
			AND (T_ExchgParam.T_Visu.T_Message.iState <> 401) THEN
		T_ExchgParam.T_Visu.T_Message.iState:=401;
	END_IF

(* Quittieren der Fehler/Warnung *)
FBResetError(	xExecute:=xExecuteResetError);
IF T_ExchgParam.T_SafetyCtrl.xResetErrorWarning THEN
	T_ExchgParam.T_SafetyCtrl.xSetForceError:=FALSE;
	CASE iStepResetError OF
		1:	xExecuteResetError:=TRUE;
			iStepResetError:=iStepResetError + 1;
		2:	IF NOT(xExecuteResetError) AND FBResetError.xDone THEN
				T_ExchgParam.T_Visu.T_Message.iState:=0;	(* Meldung löschen *)
				T_ExchgParam.T_Visu.T_Message.sDynamicTextEnglish:='';
				T_ExchgParam.T_Visu.T_Message.sDynamicTextDeutsch:='';
				T_ExchgParam.T_Visu.T_Message.sDynamicTextFrancais:='';
				T_ExchgParam.T_SafetyCtrl.xResetErrorWarning:=FALSE;
				iStepResetError:=1;
			END_IF;
	END_CASE;
ELSE
	iStepResetError:=1;
END_IF;

(* Visualisieren der Fehlermeldungen *)
RisingEdgeUpdateErrorList(CLK:=		(T_VisuQVis.T_PlcParam.dwActualPage = gT_PageNumber.iAutoMode_ErrorList) OR
								  	(T_VisuQVis.T_PlcParam.dwActualPage = gT_PageNumber.iHandMode_ErrorList) OR
								     	(T_VisuQVis.T_PlcParam.dwActualPage = gT_PageNumber.iWorkStation_ErrorList));
IF RisingEdgeUpdateErrorList.Q OR T_ExchgParam.T_SafetyCtrl.xUpdateErrorList THEN
	T_ExchgParam.T_SafetyCtrl.xUpdateErrorList:=FALSE;
	FOR ii:=1 TO 20 DO
		diErrorNr:=T_NovRAM.T_Parameter.T_ErrorNrList.adiErrorListMachine[ii];
		sErrorTimeStamp:=T_NovRAM.T_Parameter.T_ErrorNrList.asErrorTimeStampMachine[ii];
		sErrorTimeStamp:=CONCAT(sErrorTimeStamp,'--');
		IF (T_NovRAM.T_Parameter.T_ErrorNrList.asErrorTimeStampMachine[ii] <> '') THEN
			FBErrorMessageVisu(	diErrorNr:=diErrorNr ,
									T_ErrorList:=T_ErrorList);
			T_ExchgParam.T_Visu.T_MsgErrorEnglish.asMsgErrorList[ii]:=CONCAT(sErrorTimeStamp,FBErrorMessageVisu.sErrorTextEnglish);
			T_ExchgParam.T_Visu.T_MsgErrorDeutsch.asMsgErrorList[ii]:=CONCAT(sErrorTimeStamp,FBErrorMessageVisu.sErrorTextDeutsch);
		ELSE
			T_ExchgParam.T_Visu.T_MsgErrorEnglish.asMsgErrorList[ii]:='';
			T_ExchgParam.T_Visu.T_MsgErrorDeutsch.asMsgErrorList[ii]:='';
		END_IF;
	END_FOR;
END_IF;
END_PROGRAM
ACTION AxisError:
xNoProcessStationActive_St1St2:=	TProcess.T_Ctrle.xDone AND
									TStation_Work_St1.TControl.xDone AND
									(T_ExchgParam.T_Visu.T_Message.iState <> 228) AND (T_ExchgParam.T_Visu.T_Message.iState <> 229) AND (T_ExchgParam.T_Visu.T_Message.iState <> 279);
IF xNoProcessStationActive_St1St2 AND T_StartUp.T_State.xCompleted THEN
	IF RisingEdge_Station1_Axis1Error.Q THEN
		xCheckAxisError_Z_St1:=TRUE;
	END_IF;
	IF RisingEdge_Station1_Axis2Error.Q THEN
		xCheckAxisError_S_St1:=TRUE;
	END_IF;
	IF RisingEdge_Station1_Axis3Error.Q THEN
		xCheckAxisError_O_St1:=TRUE;
	END_IF;
	IF RisingEdge_Station2_Axis1Error.Q THEN
		xCheckAxisError_Z_St2:=TRUE;
	END_IF;
	IF RisingEdge_Station2_Axis2Error.Q THEN
		xCheckAxisError_S_St2:=TRUE;
	END_IF;
	IF RisingEdge_Station2_Axis3Error.Q THEN
		xCheckAxisError_O_St2:=TRUE;
	END_IF;
	IF RisingEdge_Station5_Axis1Error.Q THEN
		xCheckAxisError_C_St1:=TRUE;
	END_IF;
	TONWaitCheckError_Z_St1(IN:=xCheckAxisError_Z_St1,PT:=T#100ms);
	TONWaitCheckError_Z_St2(IN:=xCheckAxisError_Z_St2,PT:=T#100ms);
	TONWaitCheckError_S_St1(IN:=xCheckAxisError_S_St1,PT:=T#100ms);
	TONWaitCheckError_S_St2(IN:=xCheckAxisError_S_St2,PT:=T#100ms);
	TONWaitCheckError_O_St1(IN:=xCheckAxisError_O_St1,PT:=T#100ms);
	TONWaitCheckError_O_St2(IN:=xCheckAxisError_O_St2,PT:=T#100ms);
	TONWaitCheckError_C_St1(IN:=xCheckAxisError_C_St1,PT:=T#100ms);
	(* Kein Prozess und keine Station ist Aktiv, daher Eigenüberwachung der Achsen-->Überwachung nur wenn Maschine aufgestartet ist *)
	IF NOT(T_TwinSafe_Status_Z_Axis_St1.xError) AND TONWaitCheckError_Z_St1.Q AND (TStation_Work_St1.THWWorkStation.TAxisZ.T_CtrleSingle.udiErrorID <> 0) THEN
		T_ExchgParam.T_SafetyCtrl.xSetForceError:=TRUE;
		T_ExchgParam.T_SafetyCtrl.diSetForceErrorNr:=20000000 + TStation_Work_St1.THWWorkStation.TAxisZ.T_CtrleSingle.udiErrorID;
	END_IF;
	IF RisingEdge_Station1_Axis2Error.Q THEN
		T_ExchgParam.T_SafetyCtrl.xSetForceError:=TRUE;
		udi_TmpErrorNr:=	udiFct_FormatNumber(	udiNumber:=	TStation_Work_St1.THWWorkStation.TAxisS.T_CtrleSingle.udiErrorID,
													iNumberLength:=6);
		T_ExchgParam.T_SafetyCtrl.diSetForceErrorNr:=24000000 + udi_TmpErrorNr;
	END_IF;
	IF TONWaitCheckError_Z_St1.Q THEN
		xCheckAxisError_Z_St1:=FALSE;
	END_IF;
	IF TONWaitCheckError_S_St1.Q THEN
		xCheckAxisError_S_St1:=FALSE;
	END_IF;
END_IF;
END_ACTION

(* POU GENERAL/ERROR/FB_ErrorMessage, ST *)
FUNCTION_BLOCK FB_ErrorMessage
VAR_INPUT
	diErrorNr : DINT;
	T_ErrorList:ST_ERROR_LIST;
END_VAR
VAR_OUTPUT
	sErrorTextEnglish : STRING(100);
	sErrorTextDeutsch : STRING(100);
	sErrorTextFrancais : STRING(100);
END_VAR
VAR
	sTmpText1:STRING(100);
	sTmpText2:STRING(100);
	sTmpText3:STRING(100);
	sTmpText4:STRING(100);
	diTmpErrorNr:DINT;
	ptrErrorList: POINTER TO ST_LANGUAGE_LIST;
	iCounterLanguage: INT;
	sTmpErrorText : STRING(100);
	diTmpDeletePrefix: DINT;
END_VAR
(****************************************************************************************************************************************************)
(***********                     This Functionblock calculate all errors of the machine an set the follow errornumber                         ************)
(****************************************************************************************************************************************************)
ptrErrorList:=ADR(T_ErrorList.asErrorListDeutsch);	(* pointer of the errorlist, default english *)
sErrorTextEnglish:='';
sErrorTextDeutsch:='';
sErrorTextFrancais:='';
sTmpText1:='';
sTmpText2:='';
diTmpErrorNr:=0;
diTmpDeletePrefix:=0;
(* detect the error of the hardware, station or process *)
(* Fehler aus der Prozesschicht *)
(*IF iStationNr = 0 THEN sTmpText1:='Allg.Fehler: ';END_IF;*)
(* Fehler Prozesschicht *)
IF (diErrorNr < 1000000) THEN
	diTmpDeletePrefix:=0;
END_IF;
(* Fehler Stationen *)
IF (diErrorNr >= 1000000) AND (diErrorNr <= 1999999) THEN
	sTmpText1:='St1: ';
	diTmpDeletePrefix:=1000000;
END_IF;
(* Fehler von den Achsen *)
IF (diErrorNr >= 20000000) AND (diErrorNr <= 20999999) THEN
	diTmpDeletePrefix:=20000000;
	sTmpText2:='Z Achse: ';
END_IF;
IF (diErrorNr >= 24000000) AND (diErrorNr <= 24999999) THEN
	diTmpDeletePrefix:=24000000;
	sTmpText2:='S Achse: ';
END_IF;
(* Fehler von den Zylinder *)
IF (diErrorNr >= 42000000) AND (diErrorNr <= 42999999) THEN
	diTmpDeletePrefix:=42000000;
	sTmpText2:='ZylBremseZ: ';
END_IF;
(* Fehler von Prozessdaten beim schreiben auf USB-Stick *)
IF (diErrorNr >= 82000000) AND (diErrorNr <= 82999999) THEN
	diTmpDeletePrefix:=82000000;
	sTmpText2:='Prozessdaten: ';
END_IF;

FOR iCounterLanguage:=1 TO 3 DO
	sTmpText3:='';
	sTmpText4:='';
	sTmpErrorText:='';
	IF (iCounterLanguage = 1) THEN	ptrErrorList:=ADR(T_ErrorList.asErrorListDeutsch); END_IF;
	IF (iCounterLanguage = 2) THEN	ptrErrorList:=ADR(T_ErrorList.asErrorListEnglish); END_IF;
	IF (iCounterLanguage = 3) THEN	ptrErrorList:=ADR(T_ErrorList.asErrorListFrancais); END_IF;
	IF (diErrorNr >= 0) AND (diErrorNr <= 999999) THEN
		CASE diErrorNr OF
			1:		sTmpText3:=ptrErrorList^.T_LanguagList[76];		(* Not Aus Taste Maschine wurde gedrückt *)
			8:		sTmpText3:=ptrErrorList^.T_LanguagList[83];		(* Keine Druckluft *)
			9:		sTmpText3:=ptrErrorList^.T_LanguagList[100];		(* Spannungsversorgung wurde ausgeschaltet *)
			10:		sTmpText3:=ptrErrorList^.T_LanguagList[6];		(* AX5000 Parameter konnte nicht erfolgreich geschrieben werden *)		(* IGS *)
			11:		sTmpText3:=ptrErrorList^.T_LanguagList[7];		(* Achsen MasterModul2 konnte den Spindelkopf L Kanal 1 nicht finden *)	(* IGS *)
			12:		sTmpText3:=ptrErrorList^.T_LanguagList[10];		(* Achsen MasterModul2 konnte den Spindelkopf M Kanal 2 nicht finden *)	(* IGS *)
			16#F100:	sTmpText3:=ptrErrorList^.T_LanguagList[84];		(* EtherCAT 1 Klemme Fehlerhaft *)
			16#F101:	sTmpText3:=ptrErrorList^.T_LanguagList[85];		(* EtherCAT 2 Klemme Fehlerhaft *)
			16#F102:	sTmpText3:=ptrErrorList^.T_LanguagList[86];		(* Maxon EPOS nicht im Operational Mode OP *)
			16#F103:	sTmpText3:=ptrErrorList^.T_LanguagList[87];		(* SMC Ventilinsel nicht im Operational Mode OP *)
			16#F104:	sTmpText3:=ptrErrorList^.T_LanguagList[88];		(* Achsen MasterModul 1 nicht im Operational Mode OP *)
			16#F105:	sTmpText3:=ptrErrorList^.T_LanguagList[89];		(* Achsen MasterModul 2 nicht im Operational Mode OP *)				(* IGS *)
			16#F106:	sTmpText3:=ptrErrorList^.T_LanguagList[90];		(* Spannungsversorgung 24VDC fehlerhaft *)
			16#F300:	sTmpText3:=ptrErrorList^.T_LanguagList[98];		(* USB-Stick konnte nicht gefunden werden für Profil lesen/schreiben  *)
			16#F301:	sTmpText3:=ptrErrorList^.T_LanguagList[99];		(* USB-Stick konnte nicht gefunden werden für Profil löschen  *)
			16#F303:	sTmpText3:=ptrErrorList^.T_LanguagList[101];		(* Syntaxfehler mindestens einer Profildatei beim lesen aller Profile  *)
			16#F304:	sTmpText3:=ptrErrorList^.T_LanguagList[102];		(* NovRAM Speicher Fehlerhaft  *)
			16#F305:	sTmpText3:=ptrErrorList^.T_LanguagList[104];		(* USB-Stick konnte nicht gefunden werden *)
			16#F306:	sTmpText3:=ptrErrorList^.T_LanguagList[54];		(* Profil konnte nicht gespeichert werden da Verzeichnis fehlt  *)
		ELSE
			sTmpText3:=ptrErrorList^.T_LanguagList[103];	(* Nicht behandelter undefinierter Prozess Fehler *)
		END_CASE;
		IF (iCounterLanguage = 1) THEN sErrorTextDeutsch:=CONCAT(sTmpText1,sTmpText2); sErrorTextDeutsch:=CONCAT(sErrorTextDeutsch,sTmpText3); END_IF;
		IF (iCounterLanguage = 2) THEN sErrorTextEnglish:=CONCAT(sTmpText1,sTmpText2); sErrorTextEnglish:=CONCAT(sErrorTextEnglish,sTmpText3); END_IF;
		IF (iCounterLanguage = 3) THEN sErrorTextFrancais:=CONCAT(sTmpText1,sTmpText2); sErrorTextFrancais:=CONCAT(sErrorTextFrancais,sTmpText3); END_IF;
	ELSE
		IF (diErrorNr >= 1000000) AND (diErrorNr <= 4999999) THEN
			(* Gilt für Bearbeitungsstation *)
			diTmpErrorNr:=diErrorNr - diTmpDeletePrefix;
			CASE diTmpErrorNr OF
				1:	sTmpText3:=ptrErrorList^.T_LanguagList[3];	(* Z Achse-->Negativer HW Endschalter Aktiv *)
				2:	sTmpText3:=ptrErrorList^.T_LanguagList[4];	(* Z Achse-->Positiver HW Endschalter Aktiv *)
				3:	sTmpText3:=ptrErrorList^.T_LanguagList[5];	(* Z Achse-->Positiver + Negativer HW Endschalter Aktiv *)

				5:	sTmpText3:=ptrErrorList^.T_LanguagList[14];	(* Kühlmitteldruck ständig vorhanden *)
				6:	sTmpText3:=ptrErrorList^.T_LanguagList[8];	(* Kalibrierung-->ZylWzAuslenkung Sensor fehlerhaft *)
				7:	sTmpText3:=ptrErrorList^.T_LanguagList[55];	(* Kalibrierung-->ZylWzDrehmHC Sensor fehlerhaft *)
				8:	sTmpText3:=ptrErrorList^.T_LanguagList[56];	(* Kalibrierung-->ZylWzAuslenkung+ZylWzDrehmHC Sensor fehlerhaft *)
				9:	sTmpText3:=ptrErrorList^.T_LanguagList[9];	(* Z Achse muss referenziert sein *)

				11:	sTmpText3:=ptrErrorList^.T_LanguagList[59];	(* Beim starten der Bearbeitung darf DrehmSensorHCÜberlast nicht ON sein *)
				12:	sTmpText3:=ptrErrorList^.T_LanguagList[11];	(* Hubprozesslänge > Z Mech EndPos *)
				13:	sTmpText3:=ptrErrorList^.T_LanguagList[12];	(* Ausfunkhub > Z Mech EndPos *)
				14:	sTmpText3:=ptrErrorList^.T_LanguagList[13];	(* Werkzeug ist nicht im Werkstück eingefädelt *)
				15:	sTmpText3:=ptrErrorList^.T_LanguagList[29];	(* Wz Drehmoment Überlast Aktiv *)
				16:	sTmpText3:=ptrErrorList^.T_LanguagList[28];	(* Wz Drehmoment Max überschritten *)
				17:	sTmpText3:=ptrErrorList^.T_LanguagList[31];	(* Z Bearb EndPos Berechn. > Z Bearb EndPos Max *)

				18:	sTmpText3:=ptrErrorList^.T_LanguagList[33];	(* Zentrier EndPos > Z Mech EndPos *)
				19:	sTmpText3:=ptrErrorList^.T_LanguagList[34];	(* Z ZentrierPos berechn. > Z Bearb EndPos Max *)

				25:	sTmpText3:=ptrErrorList^.T_LanguagList[16];	(* Beim starten der Bearbeitung darf AuslenkSensor nicht ON sein *)
				26:	sTmpText3:=ptrErrorList^.T_LanguagList[17];	(* Beim starten der Bearbeitung darf DrehmSensorHC nicht ON sein *)
				27:	sTmpText3:=ptrErrorList^.T_LanguagList[18];	(* Z LadePos > Z Mech EndPos *)
				28:	sTmpText3:=ptrErrorList^.T_LanguagList[19];	(* Z Bearb StartPos > Z Mech EndPos *)
				29:	sTmpText3:=ptrErrorList^.T_LanguagList[20];	(* Z Bearb EndPos > Z Mech EndPos *)
				30:	sTmpText3:=ptrErrorList^.T_LanguagList[30];	(* Beim Zentrieren muss der ZylWstkEntspannen auf BearbeitPos sein *)			(* IGS3 *)
				31:	sTmpText3:=ptrErrorList^.T_LanguagList[22];	(* Z LadePos: Stimmt nicht mit anderen Positionen überein *)
				32:	sTmpText3:=ptrErrorList^.T_LanguagList[23];	(* Z Bearb StartPos: Stimmt nicht mit anderen Positionen überein *)
				33:	sTmpText3:=ptrErrorList^.T_LanguagList[24];	(* Z Bearb EndPos: Stimmt nicht mit anderen Positionen überein *)
				34:	sTmpText3:=ptrErrorList^.T_LanguagList[21];	(* Z WzWechsel Pos > Z Mech EndPos *)
				35:	sTmpText3:=ptrErrorList^.T_LanguagList[25];	(* Kalibrierung-->ZylWzAuslenkung Zylinder blockiert *)
				36:	sTmpText3:=ptrErrorList^.T_LanguagList[26];	(* Kalibrierung-->ZylWzAuslenkung Sensor fehlerhaft *)

				37:	sTmpText3:=ptrErrorList^.T_LanguagList[32];(* Z ZentrierPos berechn. > Z Mech EndPos *)


				38:	sTmpText3:=ptrErrorList^.T_LanguagList[27];	(* Kalibrierung-->ZylWzAuslenkung Zylinder blockiert *)
				39:	sTmpText3:=ptrErrorList^.T_LanguagList[57];	(* Kalibrierung-->ZylWzDrehmHC Zylinder blockiert *)
				40:	sTmpText3:=ptrErrorList^.T_LanguagList[58];	(* Kalibrierung-->ZylWzAuslenkung+ZylWzDrehmHC Zylinder blockiert *)

				41:	sTmpText3:=ptrErrorList^.T_LanguagList[60];	(* Zentrierproz. HC1 eingetroffen *)
				42:	sTmpText3:=ptrErrorList^.T_LanguagList[61];	(* Zentrierproz. StartPos erreicht und HC2 immer noch ON *)

				43:	sTmpText3:=ptrErrorList^.T_LanguagList[35];	(* Z WzZylinder Pos > Z Mech EndPos *)

				44:	sTmpText3:=ptrErrorList^.T_LanguagList[36];	(* Beim zylindrischer Teil wurde die Max EndPos erreicht  *)

				16#F101:	sTmpText3:=ptrErrorList^.T_LanguagList[48];	(* WzWechsel muss vorgenommen werden *)
				16#F220:	sTmpText3:=ptrErrorList^.T_LanguagList[1];	(* Fehler / Error während disable (Ausschalten) der Station  *)
				16#F300:	sTmpText3:=ptrErrorList^.T_LanguagList[98];	(* USB-Stick konnte nicht gefunden werden für Profil lesen/schreiben  *)
				16#F301:	sTmpText3:=ptrErrorList^.T_LanguagList[49];	(* Datei für zu ladendes Profil nicht gefunden  *)
				16#F302:	sTmpText3:=ptrErrorList^.T_LanguagList[99];	(* USB-Stick konnte nicht gefunden werden für Profil löschen  *)
				16#F303:	sTmpText3:=ptrErrorList^.T_LanguagList[51];	(* Profilname von Datei ist anders als geladenes Profil  *)
				16#F304:	sTmpText3:=ptrErrorList^.T_LanguagList[52];	(* Syntaxfehler von zu ladendes Profil  *)
				16#F305:	sTmpText3:=ptrErrorList^.T_LanguagList[102];	(* NovRAM Speicher Fehlerhaft  *)
				16#F306:	sTmpText3:=ptrErrorList^.T_LanguagList[54];	(* Profil konnte nicht gespeichert werden da Verzeichnis fehlt  *)
			ELSE
						sTmpText3:=ptrErrorList^.T_LanguagList[2];	(* Nicht behandelter undefinierter Station Fehler *)
			END_CASE;
		END_IF;

		IF (diErrorNr >= 20000000) AND (diErrorNr <= 33999999) THEN
			(* Gilt für alle Achsen *)
			diTmpErrorNr:=diErrorNr - diTmpDeletePrefix;
			CASE diTmpErrorNr OF
			(* Gilt für Beckhoff und Maxon *)
				16#F000:	sTmpText3:=ptrErrorList^.T_LanguagList[66];	(* Aufgerufene Achsfunktion besteht nicht *)
				16#F100:	sTmpText3:=ptrErrorList^.T_LanguagList[67];	(* Achsfunktion nicht ausführbar wenn Stop-Funktion Aktiv *)
				16#F501:	sTmpText3:=ptrErrorList^.T_LanguagList[109];	(* Bremse Aktiv von ST1 *)
				16#F502:	sTmpText3:=ptrErrorList^.T_LanguagList[29];	(* Wz Drehmoment Überlast Aktiv *)
			ELSE
				sTmpText3:=DINT_TO_STRING(diTmpErrorNr);
				IF (diTmpErrorNr = 16#4550) THEN
					sTmpText3:=CONCAT(sTmpText3,ptrErrorList^.T_LanguagList[75]);	(* (Schleppabstandsüberschreitung) *)
				END_IF;
			END_CASE;
		END_IF;

		IF (diErrorNr >= 40000000) AND (diErrorNr <= 77999999) THEN
			(* Gilt für alle Zylinder *)
			diTmpErrorNr:=diErrorNr - diTmpDeletePrefix;
			CASE diTmpErrorNr OF
			16#F000:		sTmpText3:=ptrErrorList^.T_LanguagList[105];	(* Zylinder Funktion nicht implementiert *)
			16#F201:		sTmpText3:=ptrErrorList^.T_LanguagList[106];	(* Zylinder Aktiv-->Sensor nicht ON *)
			16#F202:		sTmpText3:=ptrErrorList^.T_LanguagList[107];	(* Zylinder Inaktiv-->Sensor nicht ON *)
			ELSE
						sTmpText3:=ptrErrorList^.T_LanguagList[108];	(* Nicht behandelter undefinierter Zylinder Fehler *)
			END_CASE;
		END_IF;

		IF (diErrorNr >= 82000000) AND (diErrorNr <= 85999999) THEN
			(* Gilt für alle Prozessdaten *)
			diTmpErrorNr:=diErrorNr - diTmpDeletePrefix;
			CASE diTmpErrorNr OF
			201:		sTmpText3:=ptrErrorList^.T_LanguagList[146];	(* HDD steht nicht Bereit *)
			202:		sTmpText3:=ptrErrorList^.T_LanguagList[147];	(* Timeout beim Schreiben auf USB-Stick *)
			203:		sTmpText3:=ptrErrorList^.T_LanguagList[148];	(* USB Stick nicht schreibbar *)
			204:		sTmpText3:=ptrErrorList^.T_LanguagList[149];	(* USB Stick nicht gefunden *)
			END_CASE;
		END_IF;

		IF (iCounterLanguage = 1) THEN sErrorTextDeutsch:=CONCAT(sTmpText1,sTmpText2); sErrorTextDeutsch:=CONCAT(sErrorTextDeutsch,sTmpText3); END_IF;
		IF (iCounterLanguage = 2) THEN sErrorTextEnglish:=CONCAT(sTmpText1,sTmpText2); sErrorTextEnglish:=CONCAT(sErrorTextEnglish,sTmpText3); END_IF;
		IF (iCounterLanguage = 3) THEN sErrorTextFrancais:=CONCAT(sTmpText1,sTmpText2); sErrorTextFrancais:=CONCAT(sErrorTextFrancais,sTmpText3); END_IF;
	END_IF;
END_FOR;
END_FUNCTION_BLOCK

(* POU GENERAL/ERROR/FB_ResetError, ST *)
FUNCTION_BLOCK FB_ResetError
VAR_INPUT
END_VAR
VAR_IN_OUT
	xExecute:BOOL;
END_VAR
VAR_OUTPUT
	xDone:BOOL;
END_VAR
VAR
(* Trigger *)
	RisingEdgeExecute:R_TRIG;
(* Pointer *)
	ptrActivStation:POINTER TO ST_STATION;
	xFct_ResetError: BOOL;
	iStep_ResetError: INT;
	iCheckStationNr: INT;
	TONWaitReady:TON;
END_VAR
	RisingEdgeExecute(CLK:=xExecute);
	IF RisingEdgeExecute.Q THEN
	(* Init. variable by start clear error *)
		(* ...output *)
		xDone:=FALSE;
		(* ...input *)
		xExecute:=FALSE;
		xFct_ResetError:=TRUE;
		iStep_ResetError:=1;
		ptrActivStation:=ADR(TStation_Work_St1);
	END_IF;
	IF xFct_ResetError THEN
		CASE iStep_ResetError OF
			(* Überprüfe zuerst ob der Prozess im Fehlerzustand steht *)
			1:	iCheckStationNr:=1;
				IF TProcess.T_Ctrle.xEnable AND TProcess.T_Ctrle.xError THEN
					TProcess.T_Ctrle.xQuitError:=TRUE;
				ELSIF NOT(TProcess.T_Ctrle.xEnable) THEN
					TProcess.T_Ctrle.xEnable:=TRUE;
				END_IF;
				TProcess.T_Ctrle.xStop:=FALSE;
				iStep_ResetError:=iStep_ResetError + 1;
			2:	IF TProcess.T_Ctrle.xEnable AND TProcess.T_Ctrle.xDone AND NOT(TProcess.T_Ctrle.xError) AND NOT(TProcess.T_Ctrle.xQuitError) THEN
					iStep_ResetError:=iStep_ResetError + 1;
				ELSIF NOT(TProcess.T_Ctrle.xDone) AND NOT(TProcess.T_Ctrle.xError) AND NOT(TProcess.T_Ctrle.xQuitError) THEN
					TProcess.T_Ctrle.xEnable:=FALSE;
					iStep_ResetError:=1;
				END_IF;
			(* Überprüfe alle Stationen ob sie im Fehlerzustand sind *)
			3:	IF (iCheckStationNr = 1) THEN
					ptrActivStation:=ADR(TStation_Work_St1);
				ELSE
					iStep_ResetError:=iStep_ResetError + 3;	(* Aktuatoren überprüfen *)
					RETURN;
				END_IF;
				iStep_ResetError:=iStep_ResetError + 1;
			4:	IF ptrActivStation^.TControl.xEnable AND ptrActivStation^.TControl.xError THEN
					ptrActivStation^.TControl.xQuitError:=TRUE;
					iStep_ResetError:=iStep_ResetError + 1;
				ELSE
					iCheckStationNr:=iCheckStationNr + 1;	(* Nächste Station überprüfen *)
					ptrActivStation^.TControl.xQuitError:=FALSE;
					iStep_ResetError:=iStep_ResetError - 1;
				END_IF;
			5:	IF NOT(ptrActivStation^.TControl.xQuitError) AND NOT(ptrActivStation^.TControl.xError) AND ptrActivStation^.TControl.xDone THEN
					iCheckStationNr:=iCheckStationNr + 1;	(* Nächste Station überprüfen *)
					ptrActivStation^.TControl.xQuitError:=FALSE;
					iStep_ResetError:=iStep_ResetError - 2;
				END_IF;
			(* Resetten der Aktuatoren *)
			6:	IF xFct_Reset_Actuator() THEN
					TONWaitReady(IN:=FALSE);
					iStep_ResetError:=iStep_ResetError + 1;
				END_IF;
			7:	TONWaitReady(IN:=TRUE,PT:=T#0.5s);
				IF TONWaitReady.Q THEN
					iStep_ResetError:=1;
					xFct_ResetError:=FALSE;
					xDone:=TRUE;
				END_IF;
		END_CASE;
	END_IF;
END_FUNCTION_BLOCK

(* POU GENERAL/ERROR/xFct_Reset_Actuator, ST *)
FUNCTION xFct_Reset_Actuator : BOOL
VAR_INPUT
END_VAR
VAR
END_VAR
xFct_Reset_Actuator:=FALSE;
(* Resetten der Achsen *)
IF NOT(TStation_Work_St1.TControl.xResetHardware) THEN
	TStation_Work_St1.TControl.xResetHardware:=TRUE;	(* Andere Abhandlung weil Safety Drive Optionskarte im Servo intergriert ist *)
	TStation_Work_St1.TControl.xResetHardwareActivateCurrent:=TRUE;
END_IF;
(* Resetten der Zylinder *)
TStation_Work_St1.THWWorkStation.TCylBrakeReleaseZAxis.T_CtrleCyl.xReset:=TStation_Work_St1.THWWorkStation.TCylBrakeReleaseZAxis.T_CtrleCyl.xErr;
T_ProcessData_St1.T_Ctrle.xReset:=T_ProcessData_St1.T_Ctrle.xErr;
xFct_Reset_Actuator:=TRUE;
END_FUNCTION

(* POU GENERAL/ERROR/Fct_ConvertDateToString, ST *)
FUNCTION Fct_ConvertDateToString : STRING
VAR_INPUT
		iFormat:INT;	(* 0=Langes Date-Time Format; 1=Kurzes Date-Time Format; 2=Sehr Kurzes Date-Time Format *)
					(* 0='28.March 2007  08:47:01' *)
					(* 1='28.03.07 08:47' *)
					(* 2='28.03 08:47' *)
					(* 3='28.03.2007 08:47:01' *)
		TProcTimeStart:TIMESTRUCT;
END_VAR
VAR
	sTmpData:STRING(255);
	sTmpData1:STRING(255);
	wYear: WORD;
END_VAR
sTmpData:=sTmpData1:='';
IF (iFormat < 0) OR (iFormat > 3) THEN
	sTmpData1:='Wrong Date';
	Fct_ConvertDateToString:=sTmpData1;
	RETURN;
END_IF;
IF (TProcTimeStart.wDay <> 0) THEN
	IF (TProcTimeStart.wDay >= 0) AND (TProcTimeStart.wDay <= 9) THEN
		sTmpData1:=MUX(TProcTimeStart.wDay,'00','01','02','03','04','05','06','07','08','09');
		sTmpData:=CONCAT(sTmpData,sTmpData1);
	ELSE
		sTmpData:=CONCAT(sTmpData,WORD_TO_STRING(TProcTimeStart.wDay));
	END_IF;
	sTmpData:=CONCAT(sTmpData,'.');
ELSE
	sTmpData1:='Wrong Date';
	Fct_ConvertDateToString:=sTmpData1;
	RETURN;
END_IF;
IF (TProcTimeStart.wMonth <> 0) THEN
	IF (iFormat = 0) THEN
		sTmpData1:=MUX(TProcTimeStart.wMonth-1,'January','February','March','April','May','June','July','August','September','October','November','December');
	END_IF;
	IF (iFormat = 1) OR (iFormat = 2) OR (iFormat = 3) THEN
		sTmpData1:=MUX(TProcTimeStart.wMonth-1,'01','02','03','04','05','06','07','08','09','10','11','12');
	END_IF;
ELSE
	sTmpData1:='Wrong Date';
	Fct_ConvertDateToString:=sTmpData1;
	RETURN;
END_IF;
sTmpData:=CONCAT(sTmpData,sTmpData1);
IF (iFormat = 0) THEN
	sTmpData:=CONCAT(sTmpData,' ');
END_IF;
IF (iFormat = 1) THEN
	sTmpData:=CONCAT(sTmpData,'.');
END_IF;
IF (iFormat = 2) THEN
	sTmpData:=CONCAT(sTmpData,' ');
END_IF;
IF (iFormat = 3) THEN
	sTmpData:=CONCAT(sTmpData,'.');
END_IF;
IF (iFormat = 0) OR (iFormat = 1) OR (iFormat = 3) THEN
	IF (TProcTimeStart.wYear <> 0) THEN
		IF (iFormat = 0) OR (iFormat = 3) THEN
			sTmpData:=CONCAT(sTmpData,WORD_TO_STRING(TProcTimeStart.wYear));
			sTmpData:=CONCAT(sTmpData,'  ');
		END_IF;
		IF (iFormat = 1) THEN
			IF (TProcTimeStart.wYear >= 1000) AND (TProcTimeStart.wYear < 2000) THEN
				wYear:=TProcTimeStart.wYear - 1000;
			END_IF;
			IF (TProcTimeStart.wYear >= 2000) AND (TProcTimeStart.wYear < 3000) THEN
				wYear:=TProcTimeStart.wYear - 2000;
			END_IF;
			IF (wYear >= 0) AND (wYear < 10) THEN
				sTmpData1:=MUX(wYear,'00','01','02','03','04','05','06','07','08','09');
				sTmpData:=CONCAT(sTmpData,sTmpData1);
			ELSE
				sTmpData:=CONCAT(sTmpData,WORD_TO_STRING(wYear));
			END_IF;
			sTmpData:=CONCAT(sTmpData,' ');
		END_IF;
	ELSE
		sTmpData1:='Wrong Date';
		Fct_ConvertDateToString:=sTmpData1;
		RETURN;
	END_IF;
END_IF;
IF (TProcTimeStart.wHour >= 0) AND (TProcTimeStart.wHour <= 9) THEN
	sTmpData1:=MUX(TProcTimeStart.wHour,'00','01','02','03','04','05','06','07','08','09');
	sTmpData:=CONCAT(sTmpData,sTmpData1);
ELSE
	sTmpData:=CONCAT(sTmpData,WORD_TO_STRING(TProcTimeStart.wHour));
END_IF;
sTmpData:=CONCAT(sTmpData,':');
IF (TProcTimeStart.wMinute >= 0) AND (TProcTimeStart.wMinute <= 9) THEN
	sTmpData1:=MUX(TProcTimeStart.wMinute,'00','01','02','03','04','05','06','07','08','09');
	sTmpData:=CONCAT(sTmpData,sTmpData1);
ELSE
	sTmpData:=CONCAT(sTmpData,WORD_TO_STRING(TProcTimeStart.wMinute));
END_IF;
IF (iFormat = 0) OR (iFormat = 3) THEN
	sTmpData:=CONCAT(sTmpData,':');
	IF (TProcTimeStart.wSecond >= 0) AND (TProcTimeStart.wSecond <= 9) THEN
		sTmpData1:=MUX(TProcTimeStart.wSecond,'00','01','02','03','04','05','06','07','08','09');
		sTmpData:=CONCAT(sTmpData,sTmpData1);
	ELSE
		sTmpData:=CONCAT(sTmpData,WORD_TO_STRING(TProcTimeStart.wSecond));
	END_IF;
END_IF;
Fct_ConvertDateToString:=sTmpData;
END_FUNCTION

(* POU PRG_LAYER5_VISU/PRG_VISU, FBD *)
PROGRAM PRG_VISU
VAR
	FBQVIS: FBQVIS;
	FBCtrlButton: FB_CTRLEBUTTON;
	xNormalMode_EnergyON:BOOL;
	xSetupOperateA_EnergyON:BOOL;
	xSetupOperateB_EnergyON:BOOL;
	xSetupOperateC_EnergyON:BOOL;
END_VAR
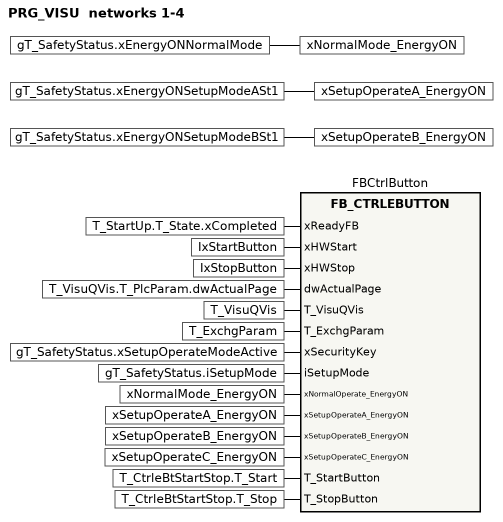
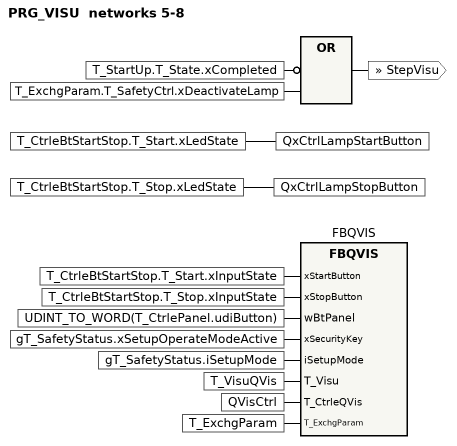
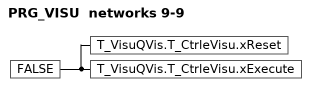
_FBD_ (* Function Block Diagram *)
NETWORK 1
	gT_SafetyStatus.xEnergyONNormalMode => xNormalMode_EnergyON
NETWORK 2
	gT_SafetyStatus.xEnergyONSetupModeASt1 => xSetupOperateA_EnergyON
NETWORK 3
	gT_SafetyStatus.xEnergyONSetupModeBSt1 => xSetupOperateB_EnergyON
NETWORK 4
	FBCtrlButton:FB_CTRLEBUTTON(xReadyFB: T_StartUp.T_State.xCompleted, xHWStart: IxStartButton, xHWStop: IxStopButton, dwActualPage: T_VisuQVis.T_PlcParam.dwActualPage, T_VisuQVis: T_VisuQVis, T_ExchgParam: T_ExchgParam, xSecurityKey: gT_SafetyStatus.xSetupOperateModeActive, iSetupMode: gT_SafetyStatus.iSetupMode, xNormalOperate_EnergyON: xNormalMode_EnergyON, xSetupOperateA_EnergyON: xSetupOperateA_EnergyON, xSetupOperateB_EnergyON: xSetupOperateB_EnergyON, xSetupOperateC_EnergyON: xSetupOperateC_EnergyON, T_StartButton: T_CtrleBtStartStop.T_Start, T_StopButton: T_CtrleBtStartStop.T_Stop)
NETWORK 5
	OR(NOT T_StartUp.T_State.xCompleted, T_ExchgParam.T_SafetyCtrl.xDeactivateLamp) => >>StepVisu
NETWORK 6
	T_CtrleBtStartStop.T_Start.xLedState => QxCtrlLampStartButton
NETWORK 7
	T_CtrleBtStartStop.T_Stop.xLedState => QxCtrlLampStopButton
NETWORK 8 StepVisu:
	FBQVIS:FBQVIS(xStartButton: T_CtrleBtStartStop.T_Start.xInputState, xStopButton: T_CtrleBtStartStop.T_Stop.xInputState, wBtPanel: UDINT_TO_WORD(T_CtrlePanel.udiButton), xSecurityKey: gT_SafetyStatus.xSetupOperateModeActive, iSetupMode: gT_SafetyStatus.iSetupMode, T_Visu: T_VisuQVis, T_CtrleQVis: QVisCtrl, T_ExchgParam: T_ExchgParam)
NETWORK 9
	FALSE => T_VisuQVis.T_CtrleVisu.xReset, T_VisuQVis.T_CtrleVisu.xExecute
_END_FBD_
(* the same logic as Structured Text *)
(* Network 1 *)
xNormalMode_EnergyON := gT_SafetyStatus.xEnergyONNormalMode;
(* Network 2 *)
xSetupOperateA_EnergyON := gT_SafetyStatus.xEnergyONSetupModeASt1;
(* Network 3 *)
xSetupOperateB_EnergyON := gT_SafetyStatus.xEnergyONSetupModeBSt1;
(* Network 4 *)
FBCtrlButton(xReadyFB := T_StartUp.T_State.xCompleted, xHWStart := IxStartButton, xHWStop := IxStopButton, dwActualPage := T_VisuQVis.T_PlcParam.dwActualPage, T_VisuQVis := T_VisuQVis, T_ExchgParam := T_ExchgParam, xSecurityKey := gT_SafetyStatus.xSetupOperateModeActive, iSetupMode := gT_SafetyStatus.iSetupMode, xNormalOperate_EnergyON := xNormalMode_EnergyON, xSetupOperateA_EnergyON := xSetupOperateA_EnergyON, xSetupOperateB_EnergyON := xSetupOperateB_EnergyON, xSetupOperateC_EnergyON := xSetupOperateC_EnergyON, T_StartButton := T_CtrleBtStartStop.T_Start, T_StopButton := T_CtrleBtStartStop.T_Stop);
(* Network 5 *)
IF NOT T_StartUp.T_State.xCompleted OR T_ExchgParam.T_SafetyCtrl.xDeactivateLamp THEN JMP StepVisu; END_IF;
(* Network 6 *)
QxCtrlLampStartButton := T_CtrleBtStartStop.T_Start.xLedState;
(* Network 7 *)
QxCtrlLampStopButton := T_CtrleBtStartStop.T_Stop.xLedState;
(* Network 8 *)
StepVisu:
FBQVIS(xStartButton := T_CtrleBtStartStop.T_Start.xInputState, xStopButton := T_CtrleBtStartStop.T_Stop.xInputState, wBtPanel := UDINT_TO_WORD(T_CtrlePanel.udiButton), xSecurityKey := gT_SafetyStatus.xSetupOperateModeActive, iSetupMode := gT_SafetyStatus.iSetupMode, T_Visu := T_VisuQVis, T_CtrleQVis := QVisCtrl, T_ExchgParam := T_ExchgParam);
(* Network 9 *)
T_VisuQVis.T_CtrleVisu.xReset := FALSE;
T_VisuQVis.T_CtrleVisu.xExecute := FALSE;
END_PROGRAM

(* POU PRG_LAYER5_VISU/FB_VISU/FBQVIS, ST *)
FUNCTION_BLOCK FBQVIS
VAR_INPUT
	xStartButton:BOOL;		(* external start button *)
	xStopButton:BOOL;		(* external stop button *)
	wBtPanel:WORD;
	xSecurityKey:BOOL;		(* state of the keyswitch-->TRUE=EinrichtBetrieb *)
	iSetupMode:INT;			(* Turn switch --> 1=EinrichtBetriebA, 2=EinrichtBetriebB, 0=Normalbetrieb *)
END_VAR
VAR_IN_OUT
	T_Visu:ST_QVIS;
	T_CtrleQVis:ST_QVISCTRLE;
	T_ExchgParam:ST_QVIS_EXCHG_PARAM;
END_VAR
VAR_OUTPUT
END_VAR
VAR
(* variable ctrle QVis*)
	xActivFB:BOOL:=FALSE;
	xConfirmResetFB:BOOL:=FALSE;
	xQvisActiv:BOOL:=FALSE;
	xChangePage:BOOL:=FALSE;
	dwInCount_QVisCmd:DWORD:=0;
	TimerQVis:TON;
	RisingEdgeExecute:R_TRIG;
	RisingEdgeActiv:R_TRIG;
	RisingEdgeReset:R_TRIG;
	iStepCount: INT;
	fbQvisInitPage:FBQVIS_INITPAGE;
	T_ConfigPage:ST_CONFIGPAGE;
	wMaskBtPanelLeft: WORD;
	wMaskBtPanelRight:WORD;
	wForceMaskBtPanelRight:WORD;
	wMaskFunctionPanel:WORD;
	wForceMaskFunctionPanel:WORD;
	aiForceRTrigActionFunctionPanel:ARRAY [1..12] OF INT;
	aiDelectRTrigActionFunctionPanel:ARRAY [1..12] OF INT;
	aiForceRTrigActionPanelRight:ARRAY [1..5] OF INT;
	aiDeleteRTrigActionPanelRight:ARRAY [1..5] OF INT;
(* variable process *)
	RisingEdgeExecuteProcess:R_TRIG;
	RisingEdgeReseTProcess:R_TRIG;
	RisingEdgeProcessDone:R_TRIG;
	RisingEdgeProcessError:R_TRIG;
	iStepProcess:INT;
	xStepProcessDone:BOOL;
	xProcessMachine: BOOL;
	xProcessStation: BOOL;
(* variable touchscreen button navigation panel panel *)
	RisingEdgeTouchScreenNavPanel:R_TRIG;
	xTmp: BOOL;
	ii: INT;
(* Key panel button "Esc"/"Enter" *)
	RisingEdgeKeyPanel_Esc:R_TRIG;
	RisingEdgeKeyPanel_Enter:R_TRIG;
(* variable start action *)
	TimerAction:TON;
	TimerNotReady:TOF;
	tTimeOutAction:TIME;
	RisingEdgeExecuteAction:R_TRIG;
	RisingEdgeResetAction:R_TRIG;
	RisingEdgeActionDone:R_TRIG;
	RisingEdgeActionNotReady:R_TRIG;
	FallingEdgeActionNotReady:F_TRIG;
	RisingEdgeActionError:R_TRIG;
	RisingEdgeTimeOut:R_TRIG;
	iStepAction:INT;
	xStepActionDone:BOOL;
	xBlockConfirmMessage: BOOL;
	xSetNewPage: BOOL;
	RisingEdgeBtPanelRight:R_TRIG;
	FallingEdgeBtPanelRight:F_TRIG;
	xPreviousPageVertical: BOOL;
	xNextPageVertical: BOOL;
	iTmp: INT;
	RisingEdgeBtPanelLeft: R_TRIG;
	xSetParameterPage: BOOL;
	xSetPreviousPage: BOOL;
	awSaveStateTaskBar: ARRAY [0..4] OF WORD;
	dwSaveActualPageTask:ARRAY [0..4,1..6] OF DWORD;
	aiTempActiveParaListState:ARRAY [0..3,1..6] OF INT;	(* 0=NormalBetrieb,1=EinrichtBetriebA,2=EinrichtBetriebB,3=EinrichtBetriebC; 1=Task1, 2=Task2..6=Task6 *)
	iSaveSetupMode:INT;
	RisingEdgeSpecialLayer: R_TRIG;
	FallingEdgeSpecialLayer: F_TRIG;
	RisingEdgeSetupMode:R_TRIG;
	iTmpSetupMode: INT;
	xForceSetupMode: BOOL;
	xForceNormalOperate: BOOL;
	TONWaitForceChangeOperateMode: TON;
	iTestCounter: INT;
	TONWaitForceChangeSetupMode: TON;
	xForceSetupOperate: BOOL;
	iTestCounter1: INT;
	RisingEdgeBtFunctionPanel: R_TRIG;
	xLampTestOnOff: BOOL;
	xLampTestBlinkOnOff: BOOL;
	xLampTestActive: BOOL;
	xLedControlButtonON: BOOL;
	xLedControlButtonOFF: BOOL;
	xLedControlLampON: BOOL;
	xLedControlLampOFF: BOOL;
	xLedSetupLampON: BOOL;
	xLedSetupLampOFF: BOOL;
	xBlinkLampAcitve: BOOL;
	iStepBlinkLampActive: INT;
	TONWaitChangeState: TON;
	iStepCheckLamp: INT;
	iPtrText: INT;
	sLineNumber: STRING;
	iStepCheckLampNumber: INT;
	iTmpPtrText: INT;
	sCopyTextLinesLampIOEngl:ARRAY [1..18] OF STRING(90);
	sCopyTextLinesLampNIOEngl:ARRAY [1..18] OF STRING(90);
	sCopyTextLinesLampIO:ARRAY [1..18] OF STRING(90);
	sCopyTextLinesLampNIO:ARRAY [1..18] OF STRING(90);
	RisingEdgeCheckLampTestPage: R_TRIG;
	wActivBtRight:WORD;
	wActivBtLeft:WORD;
	xAction_CopyProfileToProcess: BOOL;
	xProfileFileNotFoundSt1: BOOL;
	xWrongProfilNameReadedSt1: BOOL;
	xProfileFileWrongSyntaxSt1: BOOL;
	xProfileFileWrongSyntax: BOOL;
	iToLoadProfileNrSt1: INT;
	sToLoadProfileNameSt1: STRING(30);
	xAction_LoadProfile: BOOL;
	xWrongProfilNameReaded: BOOL;
	xProfileFileNotFoundSt: BOOL;
	iToLoadProfileNrSt: INT;
	sToLoadProfileNameSt: STRING(30);
	xUpdateProfileList: BOOL;
	xAction_SaveNovRAM: BOOL;
	iStepActionNovRam: INT;
(* Pointer auf die Station und HW *)
	ptrActivStation:POINTER TO ST_STATION;
	ptrActivStation_Function1:POINTER TO ST_STATION;
	ptrActivStation_FunctionStop:POINTER TO ST_STATION;
	ptrTAxisZ_St1 : POINTER TO ST_AXIS;								(* Achse für die Hubachse *)
	ptrTAxisS_St1 : POINTER TO ST_AXIS;								(* Achse für die Spindel *)

	ptrTCylToolDeflection_St1				:POINTER TO ST_CYLINDER;	(* Servoventil für das bestimmen der vertikalen Auslenkraft *)
	ptrTSensorTorque_St1 					:POINTER TO ST_CYLINDER;	(* Analoger Sensor für Drehmoment detektion *)
	ptrTCylToolTorqueHC_St1 				:POINTER TO ST_CYLINDER;	(* Drehmomentüberwachung HC *)
	ptrTCylToolTorqueOverload_St1 			:POINTER TO ST_CYLINDER;	(* Drehmomentüberwachung Überlast *)
	ptrTCylBrakeReleaseZAxis_St1 			:POINTER TO ST_CYLINDER;	(* Zylinder für lösen der Bremse bei der Z Achse *)

	ptrTCylWorkpieceClamp				:POINTER TO ST_CYLINDER;	(* Ventil für Werkstückfixierzylinder *)
	ptrTValveAirTable					:POINTER TO ST_CYLINDER;	(* Ventil für die Luft des Tisches *)
	ptrTValveVacuumTable				:POINTER TO ST_CYLINDER;	(* Ventil für die Luft des Tisches *)

	ptrTCommonAxis : POINTER TO ST_AXIS;
	ptrTCommonAxisActive		: POINTER TO ST_AXIS;
	TCommonTeachParameter:ST_EXCHG_PARAM_TEACHIN;
	ptrTCommonCylinderValve : POINTER TO ST_CYLINDER;
	ptrTCommonCylinderValveTmp : POINTER TO ST_CYLINDER;
	xAction_SaveProfile: BOOL;
	xActionDeleteProfile: BOOL;
(* activ state *)
 	T_TempActiveState:ST_TEMP_ACTIVE_STATE;
	jj: INT;
	fbCompareProfileProcessValue:FB_COMPAREPROFILEPROCESSVALUE;
	RisingEdgePtrProfileListUpDown: R_TRIG;
	iActualActiveProfile: INT;
	bOldChangeStation: BYTE;
	bOldActivStation: BYTE;
	xSetStationParameter: BOOL;
	xUpdateProfileCopyData: BOOL;
	xUpdateStationParameter: BOOL;
	RisingEdgeCheckPasswordPage: R_TRIG;
	FBPassword_SystemLevel: FB_Password_SystemLevel;
	fbGetCpuAccount:GETCPUCOUNTER;
	xChangeRandomValue: BOOL;
	RisingEdgeStandardLevel: R_TRIG;
	xChangeOperatorPassword: BOOL;
	bOldChangeSetupLevel: BYTE;
	xCylValveToggleOnOff: BOOL;
	xAxisStop: BOOL;
	xAxisTogglePower: BOOL;
	xAxisReset: BOOL;
	xAxisMoveAbsolut: BOOL;
	xAxisMoveRelative: BOOL;
	iStepActionRef: INT;
	xAxisTeachPosition: BOOL;
	xBlockSetNovRamAction_End: BOOL;
	xOnlineChange_Z_ForwardSpeedMore: BOOL;
	xOnlineChange_Z_ForwardSpeedLess: BOOL;
	xOnlineChange_Z_BackwardSpeedMore: BOOL;
	xOnlineChange_Z_BackwardSpeedLess: BOOL;
	rTmp: REAL;
	xOnlineChange_Z_BackwardOffsetMore: BOOL;
	xOnlineChange_Z_BackwardOffsetLess: BOOL;
	xOnlineChange_TorqueLevelHCMore: BOOL;
	xOnlineChange_TorqueLevelHCLess: BOOL;
	xOnlineChange_DeflectionForceMore: BOOL;
	xOnlineChange_DeflectionForceLess: BOOL;
	xOnlineChange_S_WorkSpeedMore: BOOL;
	xOnlineChange_S_WorkSpeedLess: BOOL;
	xStationWorkFunction: BOOL;
	iStationFunctionNr: INT;
	xActionProcStation: BOOL;
	xActionProcMachine: BOOL;
	xDeleteErrorList: BOOL;
	xResetErrorWarning: BOOL;
	iSaveStartedVisuFunction_St1St2: INT;
	xStationStop: BOOL;
	xProcStationStop: BOOL;
	xProcMachineStop: BOOL;
	wActivBtPanelRight: WORD;
	wTmp:WORD;
	iStationActive: INT;
	FBGetParameterList: FB_GetParameterList;
	RisingEdgeBtParameterList: R_TRIG;
	xProcessStation1ResetToolChange: BOOL;
	TONWaitReadyStartButton: TON;
	RisingEdgeCheckLampTestPage1: R_TRIG;
	RisingEdgeStartPartQualityPage: R_TRIG;
	iMessageSelected: INT:=1;
	sWrapTextEngl: STRING;
	sWrapTextGer: STRING;
	xOpenMessageWindow: BOOL;
	xCheckVisuFunctionPowerON: BOOL;
	iStepShowMessage: INT:=1;
	iSaveMessage: INT;
	TONWaitShowMessage: TON;
	xJogModeActive: BOOL;
	iStepJogModeActive: INT;
	wSaveBtPanelRight: WORD;
	xTmpJogModeActive: BOOL;
	xProcessAbordet: BOOL;
	FailingEdge_PowerSupply_NormalOperate_St1St2: F_TRIG;
	xDeleteProcessFlag_St1St2: BOOL;
	FailingEdge_PowerSupply_SetupOperateA: F_TRIG;
	xActivateLayer4_St1St2: BOOL;
	FailingEdge_PowerSupply_SetupOperateB: F_TRIG;
	xAxisMoveContinous:BOOL;
	xActivateMessage: BOOL;
	TONForceMessage: TON;
	xTmpProcMachineStop: BOOL;
	iStepActionStop: INT;
	xStepActionDoneStop: BOOL;
	xParameterButtonBlocked: BOOL;
	FBWrapWPQuality: FB_WRAP_WPQUALITY;
	xStationSetupAxisZFunction: BOOL;
	xTmpStationSetupAxisZFunction: BOOL;
	xStationSetupAxisZFunctionToolGuide: BOOL;
	xTmpStationSetupAxisZFunctionToolGuide: BOOL;
	iStepHelpVisuFunction: INT;
	xTmpStepActionDone: BOOL;
	xAxisLimitSwitchActive: BOOL;
	dwSaveVisuPage: DWORD;
	TONWaitCheckQVis: TON;
	iStepCheckQVis: INT;
	xBlockChangeVisuPage: BOOL;
	TONWaitLiftTime: TON;
	rTrigPageChanged	 :R_TRIG;
	iTmpOldPage		:DWORD;
	xNewPageInit: BOOL;
	iTmpSetupAxisSel: INT;
	xTrigAxisSelChanged: BOOL;
	xSetupPotentiometer: BOOL;
	iStepPotentiometer: INT;
	FBLinearization_Potentiometer: FB_Linearization_Potentiometer;
	xActive_Joystick: BOOL;
	xActive_EnableSwitch: BOOL;
	xReferenceState: BOOL;
	xAxisStopAll: BOOL;
	xUpdateHandlingConfig: BOOL;
	FBTeachPosToHMI:FB_TeachPosToHMI;
	rtmpAxisPosZ: REAL;
	FBGetStationFunctionNr: FB_GetStationFunctionNr;
	xInitJogVelocity: BOOL;
	lrJogVelocity: LREAL;
	xResetEnableJoystickAxisZ: BOOL;
	xSetEnableJoystickAxisZ: BOOL;
	RisingEdgeNormalMode: R_TRIG;
	RisingEdgeOperateMode: R_TRIG;
	xTriggerWait: BOOL;
	xProcessEnded: BOOL;
	sTokenString: STRING;
	FallingEdgeBtPanelLeft: F_TRIG;
	wActivBtPanelLeft: WORD;
	xDeleteProcessState: BOOL;
	xMachineDoorUpGuardControlTogOnOff: BOOL;
	xSecurityDoorUpCloseState: BOOL;
	xSecurityDoorUpOpenState: BOOL;
	xCylSetServoAnalogValue: BOOL;
	xCylPressurelessON: BOOL;
	xSpindelCalibrationONOFF: BOOL;
	rTrigButtonSt1: R_TRIG;
	rTrigButtonSt2: R_TRIG;
	rTrigButtonSt3: R_TRIG;
	rTrigButtonSt4: R_TRIG;
	xStationToolCalibrateFunction: BOOL;
	xStationSpindleBurnInFunction: BOOL;
	TONElapsedBurnInTime: TON;
	iCheckStationNr: INT;
	iStationNrReady: INT;
	iProcessFunctNr: INT;
	xStationStopWorkRight: BOOL;
	xSaveTorquePosition: BOOL;
	xSaveTorqueScale: BOOL;
	xTorqueOffsetPlus: BOOL;
	xTorqueOffsetMinus: BOOL;
	xCylTorqueOnOff: BOOL;
	xCylTorqueOverloadOnOff: BOOL;
	rZAxisSetPosition: REAL;
	TONWaitSwitchOffMessage: TON;
	xResetRockerValue: BOOL;
	xZAxisMoveToToolChangePos: BOOL;
	xZAxisMoveToLoadPos: BOOL;
(* Speichern Z EndPos Berechnet *)
	xZSaveEndPosCalc:BOOL;
	rZAxisSelectPosition: REAL;
	xSelectConfigPosition_1: BOOL;
	xSelectConfigPosition_2: BOOL;
	xSelectConfigPosition_3: BOOL;
	xSelectConfigPosition_4: BOOL;
	xSaveConfigPosition: BOOL;
	xConfigPosOnOff: BOOL;
	iSelectConfigPosition: INT;
	RisingEdgeMachineLamp: R_TRIG;
	xEndlessProcessOnOff: BOOL;

	(* .CtrlVisuFunction *)
	xCentringONOFF:BOOL;			(* IGS3 *)
	xOnlyCentringONOFF:BOOL;		(* IGS3 *)
	xSuspensionONOFF:BOOL;			(* IGS3 *)
	xCylWPUnfixONOFF:BOOL;			(* IGS3 *)

	(* .VisuFunction_SpecialFunction *)
	xRegulatorOverlaySave:BOOL;		(* IGS *)
	iTmpSelectedStationAutomat: INT;	(* IGS *)
	RisingEdgeCheckCentringProcess: R_TRIG;
	xRegulatorType1: BOOL;
	xRegulatorType2: BOOL;
	xRegulatorType3: BOOL;
	xSelectZInkWorkInfo: BOOL;
	xSelectZInkCentringInfo: BOOL;
END_VAR
ActivateFB;
IF (ABS(T_NovRam.T_Parameter.T_Machine.T_ParamSystem.iMachineNumber) < 10) THEN
	sTokenString:=CONCAT('0',INT_TO_STRING(ABS(T_NovRam.T_Parameter.T_Machine.T_ParamSystem.iMachineNumber)));
ELSIF (ABS(T_NovRam.T_Parameter.T_Machine.T_ParamSystem.iMachineNumber) < 100) THEN
	sTokenString:=INT_TO_STRING(ABS(T_NovRam.T_Parameter.T_Machine.T_ParamSystem.iMachineNumber));
ELSE
	sTokenString:='00';
END_IF;
T_ExchgParam.T_Visu.sQVisVersion:=CONCAT(T_ExchgParam.T_Visu.sSWVersion,sTokenString);
T_ExchgParam.T_Visu.sHWVersion:=CONCAT(T_ExchgParam.T_Visu.sSWVersion,sTokenString);

gxBlockChangeMovementVisuActiveMessage:=	xProcessStation OR xProcessMachine OR xStationSetupAxisZFunction OR xTmpStationSetupAxisZFunction OR xStationSetupAxisZFunctionToolGuide OR xTmpStationSetupAxisZFunctionToolGuide;

(* Exit FB if FB desactiv *)
	IF NOT(xActivFB)  THEN
		RETURN;
	END_IF
ResetVisu;
InitQVis;
(* exit FB if Qvis inactiv *)
IF NOT(T_Visu.T_CtrleVisu.xQvis) THEN RETURN; END_IF
(* Check UPS Power fail *)
IF T_CtrleUPS.xBlockSystem_PowerFail THEN RETURN; END_IF;
(* Monitor dynamic mask for button panel right and function panel *)
IF T_Visu.T_CtrleProcess.xDone OR T_Visu.T_CtrleProcess.xErr THEN
(* Set the standard mask *)
	wMaskBtPanelLeft:=T_ConfigPage.wMaskBtPanelLeft;
	wMaskBtPanelRight:=T_ConfigPage.wMaskBtPanelRight;
	wMaskFunctionPanel:=T_ConfigPage.wMaskFunctionPanel;
(* Set the dynamic mask *)
ELSE	wMaskBtPanelLeft:=T_ConfigPage.wMaskBtPanelLeft AND T_ConfigPage.wMaskProcBtPanelLeft;
		IF (T_ExchgParam.T_Visu.T_Message.iState <> 401) THEN
			wMaskBtPanelRight:=T_ConfigPage.wMaskProcBtPanelRight;
		ELSE
			wMaskBtPanelRight:=T_ConfigPage.wMaskBtPanelRight;	(* Fehler muss quittiert werden können *)
		END_IF;
		wMaskFunctionPanel:=T_ConfigPage.wMaskProcFunctionPanel;
END_IF
(* Update Page configuration *)
IF (T_Visu.T_PlcParam.dwActualPage >= 1) AND (T_Visu.T_PlcParam.dwActualPage <= 999) THEN
	T_ConfigPage:=T_Visu.T_ConfigPage[T_Visu.T_PageIndex[T_Visu.T_PlcParam.dwActualPage].iIndexConfigPage];
END_IF;
(* Config. divers mask *)
T_ExchgParam.T_TouchScreenBtPanel.iNotMaskTextBt
	:=(16#1F XOR wMaskBtPanelLeft) OR (16#3E0 XOR wMaskBtPanelRight);
IF xParameterButtonBlocked THEN
	T_ExchgParam.T_TouchScreenBtPanel.iNotMaskTextBt:=WORD_TO_INT(INT_TO_WORD(T_ExchgParam.T_TouchScreenBtPanel.iNotMaskTextBt) OR 16#10);	(* Falls Zugang zu Parameter gesperrt ist, dann wird die Anzeige für die Parameterebene gesperrt *)
END_IF;
(* management Fn button panel availability *)
T_ExchgParam.T_BtFunctionPanel.wNotMasktext:=16#FFF XOR wMaskFunctionPanel;
(* management navigation panel mask *)
T_ExchgParam.T_TouchScreenNavPanel.wNotMasktext:=T_ConfigPage.wMaskTouchScreenNavPanel;
T_ExchgParam.T_TouchScreenBtPanel.iStateBtLeft:=iFct_GetLeftButtonNumber(dwActualPage:=T_Visu.T_PlcParam.dwActualPage);
IF xFct_GetParameterPageActive(dwActualPage:=T_Visu.T_PlcParam.dwActualPage) THEN
	T_ExchgParam.T_TouchScreenNavPanel.wState:=awSaveStateTaskBar[T_ExchgParam.T_Visu.bActiveSetupMode];
ELSE
	T_ExchgParam.T_TouchScreenNavPanel.wState:=wFct_GetTaskNumber(dwActualPage:=T_Visu.T_PlcParam.dwActualPage);
END_IF;
T_ExchgParam.T_Visu.iHeaderTitlePageNumber:=DWORD_TO_INT(T_Visu.T_PlcParam.dwActualPage);
IF gT_SafetyStatus.xSetupOperateModeActive THEN
	IF (T_ExchgParam.T_TouchScreenBtPanel.iStateBtLeft >= 16) THEN
		T_ExchgParam.T_Visu.bActiveSetupMode:=INT_TO_BYTE(iFct_GetBitNumber(wInputButton:=INT_TO_BYTE(T_ExchgParam.T_TouchScreenBtPanel.iStateBtLeft - 16)));
	ELSE
		T_ExchgParam.T_Visu.bActiveSetupMode:=INT_TO_BYTE(iFct_GetBitNumber(wInputButton:=INT_TO_BYTE(T_ExchgParam.T_TouchScreenBtPanel.iStateBtLeft)));
	END_IF;
ELSE
	T_ExchgParam.T_Visu.bActiveSetupMode:=0;
END_IF;
xFct_SetActualPageTask(	dwActualPage:=T_Visu.T_PlcParam.dwActualPage,
							iTaskBarNumber:=(iFct_GetBitNumber(wInputButton:=T_ExchgParam.T_TouchScreenNavPanel.wState)),
							dwSaveActualPageTask:=dwSaveActualPageTask);
IF T_ExchgParam.T_Config.xNoTouchScreenBtPanel THEN
	wActivBtLeft:=wBtPanel AND 16#1F;
	wActivBtRight:=wBtPanel AND 16#3E0;
ELSE
	wActivBtLeft:=INT_TO_WORD(T_ExchgParam.T_TouchScreenBtPanel.iActivBtLeft);
	wActivBtRight:=INT_TO_WORD(T_ExchgParam.T_TouchScreenBtPanel.iActivBtRight);
END_IF;
TONWaitReadyStartButton(IN:=TRUE,PT:=T#1s);
IF T_StartUp.T_State.xCompleted THEN
	CtrlSetupKeySwitch;
	CtrlSetupOperateModeSwitch;
END_IF;
CheckSecurityDeactivate;
CtrlPanelLeftButton;
CtrlPanelRightButton;
CtrlParaListButton;
CtrlTaskBar;
CtrlFunctionButton;
CtrlStartStopButton;
CtrlSpindleTime;
MaskFunctionButton;
MaskRightButton;
Monitor_FctButton_Led;
UserLevel;
VisuUpdateParameter;
Monitor_Station;
ChangeStation;
Monitor_ActuatorState;
Monitor_Function;
ChangeWPQuality;
ProfileManagement;
CtrlVisuFunction;
VisuFunction_SetNewPageVertical;
VisuFunction_SetNewPage;
VisuFunction_SetParameterPage;
VisuFunction_SetPreviousPage;
VisuFunction_ErrorManagement;
VisuFunction_LampTest;
VisuFunction_MachineLamp;
VisuFunction_SetupPotentiometer;
VisuFunction_SetupTorque;
VisuFunction_SafetyDoor;
VisuFunction_ChangePassword;
VisuFunction_OnlineChange;
VisuFunction_Axis;
VisuFunction_AxisTeach;
VisuFunction_CylinderValve;
VisuFunction_StationStop;
VisuFunction_StationFunction;
VisuFunction_ToolChange;
VisuFunction_ToolCalibration;
VisuFunction_SpindleBurnIn;
VisuFunction_Setup_Z_Axis;
VisuFunction_Setup_Z_Axis_ToolGuide;
VisuFunction_SpecialFunction;
VisuFunction_ProcessState;
VisuFunction_ProcessStop;
VisuFunction_ProcessFunction;
VisuFunction_NovRAM;
VisuFunction_ProfileManagement;
CtrlProcessFunction;
CtrlPreWarning;
ChangeVisuPage;
T_ExchgParam.T_BtFunctionPanel.wActivBt:=0;
IF NOT(xTmpStationSetupAxisZFunction) AND NOT(xTmpStationSetupAxisZFunctionToolGuide) THEN
	gxSetupFunctionActive:=FALSE;
END_IF;
IF NOT(xAxisMoveAbsolut) AND NOT(xZAxisMoveToToolChangePos) AND NOT(xZAxisMoveToLoadPos) THEN
	gxAxisAbsolutMovementActive:=FALSE;
END_IF;

(* IGS wenn eine Overlay MessageBox aktiv ist: xMessageActive setzen *)
T_ExchgParam.T_SafetyCtrl.xMessageActive:=	(T_ExchgParam.T_SafetyCtrl.bStateMessageError<>0)
											OR (T_ExchgParam.T_SafetyCtrl.bStateMessageInfo<>0)
											OR (T_ExchgParam.T_SafetyCtrl.bStateMessagePreWarning<>0)
											OR (T_ExchgParam.T_SafetyCtrl.bStateMessageRequest<>0)
											OR (T_ExchgParam.T_SafetyCtrl.bStateMessageWarning<>0);
END_FUNCTION_BLOCK
ACTION ActivateFB:
	RisingEdgeActiv(	CLK:=T_Visu.T_CtrleVisu.xActive);
	IF RisingEdgeActiv.Q THEN
		(* call functionblock init. *)
		fbQvisInitPage(	T_Visu:=T_Visu);
		(* Init. variable for visualisation action *)
		T_Visu.T_CtrleAction.xDone:=TRUE;
		T_Visu.T_CtrleAction.xNotReady:=FALSE;
		T_Visu.T_CtrleAction.xErr:=FALSE;
		T_Visu.T_CtrleAction.udiErrorID:=0;
		(* Initialisieren der Pointer der Station und Hardware *)
		ptrActivStation:=ADR(TStation_Work_St1);
		ptrTAxisZ_St1:=ADR(TStation_Work_St1.THWWorkStation.TAxisZ);
		ptrTAxisS_St1:=ADR(TStation_Work_St1.THWWorkStation.TAxisS);

		ptrTSensorTorque_St1						:=ADR(TStation_Work_St1.THWWorkStation.TSensorTorque);
		ptrTCylToolDeflection_St1					:=ADR(TStation_Work_St1.THWWorkStation.TCylToolDeflection);
		ptrTCylBrakeReleaseZAxis_St1 				:=ADR(TStation_Work_St1.THWWorkStation.TCylBrakeReleaseZAxis);

		ptrTCylToolTorqueHC_St1					:=ADR(TStation_Work_St1.THWWorkStation.TCylToolTorqueHC);
		ptrTCylToolTorqueOverload_St1				:=ADR(TStation_Work_St1.THWWorkStation.TCylToolTorqueOverload);
		ptrTCylWorkpieceClamp						:=ADR(TStation_Work_St1.THWWorkStation.TCylWorkpieceClamp);
		ptrTValveAirTable							:=ADR(TStation_Work_St1.THWWorkStation.TValveAirTable);
		ptrTValveVacuumTable						:=ADR(TStation_Work_St1.THWWorkStation.TValveVacuumTable);

		ptrTCommonAxis:=ADR(TStation_Work_St1.THWWorkStation.TAxisZ);
		ptrTCommonAxisActive	:=ADR(TStation_Work_St1.THWWorkStation.TAxisZ);

		ptrTCommonCylinderValve:=ADR(TStation_Work_St1.THWWorkStation.TCylToolDeflection);
		ptrTCommonCylinderValveTmp:=ADR(TStation_Work_St1.THWWorkStation.TCylToolDeflection);

		(* Init. Temporary active state for station 1 to 3 *)
		T_TempActiveState.iActValve_SetupB1_St1:=5;
		T_TempActiveState.iActAxis_SetupB1_St1:=1;
		T_TempActiveState.iActCyl_SetupB1_St1:=1;
		T_TempActiveState.iActCylinderSetup_SetupB1:=2;
		T_TempActiveState.iActiveProfile:=1;
		T_TempActiveState.iPtrListProfile:=1;
		iActualActiveProfile:=-1;
		FOR ii:=1 TO 5 DO
			T_ExchgParam.T_ProfileCommon.T_ProfileList[ii].iNumber:=ii;
			T_ExchgParam.T_ProfileCommon.T_ProfileList[ii].sName:='';
		END_FOR
		(* init. variable *)
		T_ExchgParam.T_FunctionCommon.iFunctionNrMicrohead:=1;
		T_ExchgParam.T_TouchScreenBtPanel.iSelectStationNumber:=1;
		T_ExchgParam.T_StationCommon.bSelectCylinderConfig:=1;
		T_ExchgParam.T_StationCommon.bSelectZAxisProcedure:=1;
		T_ExchgParam.T_StationCommon.iSelectConfigPosition:=1;
		iSelectConfigPosition:=1;
		T_ExchgParam.T_Visu.bActivStation:=1;
		bOldChangeStation:=16#FF;
		bOldChangeSetupLevel:=16#FF;
		bOldActivStation:=1;
		T_ExchgParam.T_Visu.T_Level.iActLevel:=0;
		T_ExchgParam.T_Visu.T_Level.diPwUser:=-1;
		T_ExchgParam.T_Visu.T_Level.diPwOperator:=-1;
		T_ExchgParam.T_Visu.T_Level.diPwSystem:=-1;
		T_ExchgParam.T_StationCommon.xBlockSelectAutoMode:=FALSE;
		TONWaitCheckQVis(IN:=FALSE);
		(* set activation *)
		xActivFB:=TRUE;
		gxSpindelCalibrationONOFF_St1:=TRUE;
		T_ExchgParam.T_StationCommon.bSelectShowIncValue:=0;
	END_IF;
END_ACTION
ACTION ChangeStation:
IF T_StartUp.T_State.xCompleted THEN
	RisingEdgeNormalMode(CLK:=NOT(gT_SafetyStatus.xSetupOperateModeActive));
	RisingEdgeOperateMode(CLK:=gT_SafetyStatus.xSetupOperateModeActive);
	IF RisingEdgeNormalMode.Q OR RisingEdgeOperateMode.Q THEN
		xSetStationParameter:=TRUE;
	END_IF;
END_IF;
IF xSetStationParameter OR rTrigButtonSt1.Q OR rTrigButtonSt2.Q OR rTrigButtonSt3.Q OR rTrigButtonSt4.Q THEN
	xSetStationParameter:=FALSE;
	(* Update display  list *)
	xUpdateProfileList:=TRUE;
	(* Update display copy data *)
	xUpdateProfileCopyData:=TRUE;
	xUpdateStationParameter:=TRUE;
END_IF;
IF xUpdateStationParameter THEN
	xUpdateStationParameter:=FALSE;
	T_ExchgParam.T_StationCommon.T_Param_Machine.T_ParamSystem:=T_NovRAM.T_Parameter.T_Machine.T_ParamSystem;
	T_ExchgParam.T_StationCommon.T_Param_Machine.adiPotentiometerValue:=T_NovRAM.T_Parameter.T_Machine.adiPotentiometerValue;
	T_ExchgParam.T_StationCommon.T_ToolCounter_St1:=T_NovRam.T_Parameter.T_StationWork[gciStationSt1].T_ToolCounter;
	T_ExchgParam.T_StationCommon.T_WPCounter_St1:=T_NovRam.T_Parameter.T_StationWork[gciStationSt1].T_WPCounter;
	T_ExchgParam.T_StationCommon.T_Param_StationWork:=T_NovRam.T_Parameter.T_StationWork[gciStationSt1];
	IF T_StartUp.T_State.xCompleted THEN
		T_ExchgParam.T_ProfileCommon.T_Id.iNumber:=T_NovRam.T_Parameter.T_StationWork[gciStationSt1].T_InfoProcess.iProfile;
		T_ExchgParam.T_ProfileCommon.T_Id.sName:=T_NovRam.T_Parameter.T_StationWork[gciStationSt1].T_InfoProcess.sProfileName;
	END_IF;
	T_ExchgParam.T_SpindleBurnIn.rTimeActive:=T_NovRAM.T_Parameter.T_StationWork[gciStationSt1].T_Fct_SpindleBurnIn.rTimeSpindleActive;
	T_ExchgParam.T_SpindleBurnIn.rTimeInactive:=T_NovRAM.T_Parameter.T_StationWork[gciStationSt1].T_Fct_SpindleBurnIn.rTimeSpindleInactive;
	T_ExchgParam.T_SpindleBurnIn.rTimeMaxActiveFunction:=T_NovRAM.T_Parameter.T_StationWork[gciStationSt1].T_Fct_SpindleBurnIn.rTimeMaxActiveFunction;
	T_ExchgParam.T_SpindleBurnIn.rSpeed_Axis_S:=T_NovRAM.T_Parameter.T_StationWork[gciStationSt1].T_Fct_SpindleBurnIn.rSpindleSpeed;
	CASE T_ExchgParam.bToolSpindleActive OF
	1:	(* Maxon Spindel *)
		T_ExchgParam.T_AnalogSensTorque.rMeasureDistance:=T_NovRAM.T_Parameter.T_StationWork[gciStationSt1].T_TorqueSystem.rMeasureDistance;
		T_ExchgParam.T_AnalogSensTorque.rScaleFactor:=T_NovRAM.T_Parameter.T_StationWork[gciStationSt1].T_TorqueSystem.rTorqueScaleFactor;
	2,3:	(* Beckhoff Spindel *)
		T_ExchgParam.T_AnalogSensTorque.rMeasureDistance:=0;
		T_ExchgParam.T_AnalogSensTorque.rScaleFactor:=0;
	END_CASE;
	IF (T_Visu.T_PlcParam.dwActualPage = gT_PageNumber.iHandMode_Parameter)  AND (T_ExchgParam.T_BtParameterList.iEditParam <> 117) AND (T_Visu.T_PlcParam.dwActualPage <> gT_PageNumber.iWorkStation_Axis1) THEN
		T_ExchgParam.T_StationCommon.rPositionEndProcCalc:=garPositionEndProcCalc[1];
		T_ExchgParam.T_StationCommon.rCentringEndProcCalc:=garCentringEndProcCalc[1];
	END_IF;

END_IF;
(*Detect Page changed?*)
rTrigPageChanged(CLK:=iTmpOldPage <>T_Visu.T_PlcParam.dwActualPage);
iTmpOldPage:=T_Visu.T_PlcParam.dwActualPage;

IF rTrigPageChanged.Q THEN
	T_ExchgParam.T_BtFunctionPanel.wState:=0;(*Fxx->inaktiv*)
	xUpdateStationParameter:=TRUE;
	 xNewPageInit:=FALSE;
	xUpdateHandlingConfig:=TRUE;
END_IF
(* Nach Seitenwechsel:  Init Anwahl Achse oder Zylinder und Funktionsauswahl pro EinrichtSeite:*)
CASE T_Visu.T_PlcParam.dwActualPage OF
gT_PageNumber.iWorkStation_Axis1:
	IF rTrigPageChanged.Q THEN
		T_ExchgParam.T_TeachIn.iSetup_AxisSel:=T_TempActiveState.iActAxis_SetupB1_St1;
	END_IF
	IF (T_TempActiveState.iActAxis_SetupB1_St1 <> T_ExchgParam.T_TeachIn.iSetup_AxisSel) THEN
		T_TempActiveState.iActAxis_SetupB1_St1:=T_ExchgParam.T_TeachIn.iSetup_AxisSel;
	END_IF;
	IF (T_ExchgParam.T_TeachIn.iSetup_AxisSel = 2) THEN
		CASE T_ExchgParam.bToolSpindleActive OF
		2,3:	T_ExchgParam.T_TeachIn.iSetup_AxisSel:=3;
		END_CASE;
	END_IF;

gT_PageNumber.iWorkStation_Cylinder1:
	IF rTrigPageChanged.Q THEN
		T_ExchgParam.T_Cylinder.iSelCyl_Setup:=T_TempActiveState.iActCyl_SetupB1_St1;
	END_IF
	IF (T_TempActiveState.iActCyl_SetupB1_St1 <> T_ExchgParam.T_Cylinder.iSelCyl_Setup) THEN
		T_TempActiveState.iActCyl_SetupB1_St1:=T_ExchgParam.T_Cylinder.iSelCyl_Setup;
	END_IF;

gT_PageNumber.iWorkStation_Valve1:
	IF rTrigPageChanged.Q THEN
		T_ExchgParam.T_Cylinder.iSelCyl_Setup:=T_TempActiveState.iActValve_SetupB1_St1;
	END_IF
	IF (T_TempActiveState.iActValve_SetupB1_St1 <> T_ExchgParam.T_Cylinder.iSelCyl_Setup) THEN
		T_TempActiveState.iActValve_SetupB1_St1:=T_ExchgParam.T_Cylinder.iSelCyl_Setup;
	END_IF;

gT_PageNumber.iWorkStation_Setup4:
	IF rTrigPageChanged.Q THEN
		T_ExchgParam.T_Cylinder.iSelCyl_Setup:=T_TempActiveState.iActCylinderSetup_SetupB1;
	END_IF
	IF (T_TempActiveState.iActCylinderSetup_SetupB1 <> T_ExchgParam.T_Cylinder.iSelCyl_Setup) THEN
		T_TempActiveState.iActCylinderSetup_SetupB1:=T_ExchgParam.T_Cylinder.iSelCyl_Setup;
	END_IF;
END_CASE;
(*Check for Axis Selection Change*)
xTrigAxisSelChanged:=iTmpSetupAxisSel <>T_ExchgParam.T_TeachIn.iSetup_AxisSel OR rTrigPageChanged.Q;
iTmpSetupAxisSel:=T_ExchgParam.T_TeachIn.iSetup_AxisSel;
IF xTrigAxisSelChanged THEN (*Init Value at Selection change*)
	T_ExchgParam.T_TeachIn.arAxis[gciAxisZ_St1].rSetPos:=TStation_Work_St1.THWWorkStation.TAxisZ.T_LiveValue.lrActualPosition;
END_IF
(* Zuweisen der Datenstruktur der ausgewählten Achse *)
IF (T_Visu.T_PlcParam.dwActualPage =  gT_PageNumber.iWorkStation_Axis1) THEN
	CASE  T_ExchgParam.T_TeachIn.iSetup_AxisSel   OF
		1:	(*1=Z Achse *)
			ptrTCommonAxis:=ptrTAxisZ_St1;
			TCommonTeachParameter:=gcarAxisConfig[gciAxisZ_St1];
			ptrTCommonAxis^.T_CtrleSingle.xSlowFast:=FALSE;
			ptrTCommonAxis^.T_CtrleSingle.xJogInc:=T_ExchgParam.T_TeachIn.xJogInc_Common_Setup_Axis;
			IF T_ExchgParam.T_TeachIn.arAxis[gciAxisZ_St1].iTeachSelPos = 0 THEN(*eingabe-Wertt*)
				TCommonTeachParameter.rRefPosition:=
				T_ExchgParam.T_TeachIn.arAxis[gciAxisZ_St1].rSetPos ;
			ELSE(*oder gespeicherter Wert, siehe MonitorActuatorState*)
				TCommonTeachParameter.rRefPosition:=
				T_ExchgParam.T_TeachIn.arAxis[gciAxisZ_St1].rTeachPosStored;
			END_IF
		2,3:	(*2 & 3=S Achse *)
			ptrTCommonAxis:=ptrTAxisS_St1;
			TCommonTeachParameter:=gcarAxisConfig[gciAxisS_St1];
			ptrTCommonAxis^.T_CtrleSingle.xSlowFast:=FALSE;
			ptrTCommonAxis^.T_CtrleSingle.xJogInc:=T_ExchgParam.T_TeachIn.xJogInc_Common_Setup_Axis;
			TCommonTeachParameter.rPositionSpeed:=
				T_ExchgParam.T_TeachIn.arAxis[gciAxisS_St1].rSetSpeed;
	END_CASE
END_IF;

(* Zuweisen der Datenstruktur der ausgewählten Zylinder oder Ventile *)
IF (T_Visu.T_PlcParam.dwActualPage =  gT_PageNumber.iWorkStation_Cylinder1) OR
    (T_Visu.T_PlcParam.dwActualPage =  gT_PageNumber.iWorkStation_Valve1) OR
    (T_Visu.T_PlcParam.dwActualPage =  gT_PageNumber.iWorkStation_Setup4) THEN
	CASE  T_ExchgParam.T_Cylinder.iSelCyl_Setup   OF
(*
01	Zylinder-->Wz Auslenkung
02	Zylinder-->Wz Drehmoment HC
03	Zylinder-->Wz Drehmoment Überl.
04	Zylinder-->Bremse Z Achse
05	Zylinder-->Wstk Spannung
06	Ventil-->Luft Tisch
07	Ventil-->Vakuum Tisch*)
		1:	ptrTCommonCylinderValve:=ptrTCylToolDeflection_St1;
		2:	ptrTCommonCylinderValve:=ptrTCylToolTorqueHC_St1;
		3:	ptrTCommonCylinderValve:=ptrTCylToolTorqueOverload_St1;
		4:	ptrTCommonCylinderValve:=ptrTCylBrakeReleaseZAxis_St1;
		5:	ptrTCommonCylinderValve:=ptrTCylWorkpieceClamp;
		6:	ptrTCommonCylinderValve:=ptrTValveAirTable;
		7:	ptrTCommonCylinderValve:=ptrTValveVacuumTable;
	END_CASE
END_IF

IF T_StartUp.T_State.xCompleted THEN
	T_ExchgParam.T_StationCommon.T_Param_StationWork.T_InfoProcess:=T_NovRam.T_Parameter.T_StationWork[gciStationSt1].T_InfoProcess;
	T_ExchgParam.T_TeachIn.arAxisCommon.rActPos:=										TStation_Work_St1.THWWorkStation.TAxisZ.T_LiveValue.lrActualPosition;
	T_ExchgParam.T_TeachIn.arAxisCommon.rActSpeed:=										TStation_Work_St1.THWWorkStation.TAxisZ.T_LiveValue.lrActualVelocity;
	T_ExchgParam.T_TeachIn.rAxisSSpeedCommon:=											TStation_Work_St1.THWWorkStation.TAxisS.T_LiveValue.lrActualVelocity;

	IF NOT(xSecurityKey) THEN
		T_ExchgParam.T_StationCommon.T_Param_StationWork.T_InfoProcess:=						T_NovRam.T_Parameter.T_StationWork[gciStationSt1].T_InfoProcess;
		T_ExchgParam.T_StationCommon.T_Param_StationWork.T_InfoProcess.iHCTorquePos:=		TStation_Work_St1.THWWorkStation.TCtrlWork.iHCTorquePos;
		T_ExchgParam.T_StationCommon.T_Param_StationWork.T_InfoProcess.iHCDeflectionPos:=		TStation_Work_St1.THWWorkStation.TCtrlWork.iHCDeflectionPos;

		IF NOT(xFct_GetParameterPageActive(dwActualPage:=T_Visu.T_PlcParam.dwActualPage)) THEN
			T_ExchgParam.T_StationCommon.T_Param_StationWork.T_WPCounter:=T_NovRAM.T_Parameter.T_StationWork[gciStationSt1].T_WPCounter;
			T_ExchgParam.T_StationCommon.T_Param_StationWork.T_ToolCounter:=T_NovRam.T_Parameter.T_StationWork[gciStationSt1].T_ToolCounter;
		END_IF;
	END_IF;
END_IF;
END_ACTION
ACTION ChangeVisuPage:
(* waiting for changing page *)
	RisingEdgeExecute(CLK:=T_Visu.T_CtrleVisu.xExecute);
	IF RisingEdgeExecute.Q THEN
		iStepCount:=iStepCount + 1;
		CASE T_Visu.T_CtrleVisu.iFunction OF
		(* change page *)
		1:	xChangePage:=TRUE;
			dwInCount_QVisCmd:=T_CtrleQVis.dwInCount;
		ELSE
		(* function not implemented *)
			T_Visu.T_CtrleVisu.xDone:=FALSE;
			T_Visu.T_CtrleVisu.xErr:=TRUE;
			T_Visu.T_CtrleVisu.udiErrorID:=16#F000;
		END_CASE
		(* Init. variable *)
		T_Visu.T_CtrleVisu.xDone:=FALSE;
		T_Visu.T_CtrleVisu.xErr:=FALSE;
		T_Visu.T_CtrleVisu.udiErrorID:=0;
		(* exit FB *)
		RETURN;
	END_IF

(* waiting for changing page from the PLC *)
	IF xChangePage AND NOT(xBlockChangeVisuPage) THEN
		IF dwInCount_QVisCmd = T_CtrleQVis.dwInCount THEN
			(* Init. command *)
			T_CtrleQVis.dwInCommand:=1;
			T_CtrleQVis.dwInQVisCtrlAddress:=ADR(T_CtrleQVis);
			T_CtrleQVis.dwInParameterAddress:=ADR(T_Visu.T_PlcParam.dwSetNewPage);
			(* start command *)
			T_CtrleQVis.dwInCount:=T_CtrleQVis.dwInCount+1;
		ELSE
			IF T_CtrleQVis.dwInCount = T_CtrleQVis.dwOutCount THEN
			(* command done *)
				T_Visu.T_CtrleVisu.xExecute:=FALSE;
				IF T_CtrleQVis.diOutStatus = 0 THEN
				(* command done without error *)
					T_Visu.T_CtrleVisu.xDone:=TRUE;
					T_Visu.T_CtrleVisu.xErr:=FALSE;
					T_Visu.T_CtrleVisu.udiErrorID:=0;
					T_Visu.T_PlcParam.dwPreviousPage:=T_Visu.T_PlcParam.dwActualPage;
					T_Visu.T_PlcParam.dwActualPage:=T_Visu.T_PlcParam.dwSetNewPage;
					T_ExchgParam.T_Visu.T_Message.iState:=0;
				ELSE
				(* command done with error *)
					T_Visu.T_CtrleVisu.xDone:=FALSE;
					T_Visu.T_CtrleVisu.xErr:=TRUE;
					T_Visu.T_CtrleVisu.udiErrorID:=16#F400 + DINT_TO_UDINT(T_CtrleQVis.diOutStatus);
				END_IF
				(* reset variable 'xChangePage' *)
				xChangePage:=FALSE;
			END_IF
		END_IF
	END_IF
END_ACTION
ACTION ChangeWPQuality:
RisingEdgeStartPartQualityPage(CLK:=(T_Visu.T_PlcParam.dwActualPage = gT_PageNumber.iAutoMode_PartQuality));
IF (T_Visu.T_PlcParam.dwActualPage = gT_PageNumber.iAutoMode_PartQuality) THEN

(* Auswahl des Wstk für die Analyse *)
(* Part Quality *)


	IF T_ExchgParam.T_StationCommon.T_Button_Quality_Backward.xActive THEN
		T_ExchgParam.T_StationCommon.T_Button_Quality_Backward.xActive:=FALSE;
		T_ExchgParam.T_StationCommon.T_Input_Quality_HoleNumber.diInput1:=T_ExchgParam.T_StationCommon.T_Input_Quality_HoleNumber.diInput1 - 1;
		IF (T_ExchgParam.T_StationCommon.T_Input_Quality_HoleNumber.diInput1 < T_NovRam.T_Parameter.T_PartAnalysis[gciStationSt1].adiNumberHole[1]) THEN
			T_ExchgParam.T_StationCommon.T_Input_Quality_HoleNumber.diInput1:=T_NovRam.T_Parameter.T_PartAnalysis[gciStationSt1].adiNumberHole[1];
		END_IF;
	END_IF;
	IF T_ExchgParam.T_StationCommon.T_Button_Quality_Forward.xActive THEN
		T_ExchgParam.T_StationCommon.T_Button_Quality_Forward.xActive:=FALSE;
		T_ExchgParam.T_StationCommon.T_Input_Quality_HoleNumber.diInput1:=T_ExchgParam.T_StationCommon.T_Input_Quality_HoleNumber.diInput1 + 1;
		IF (T_ExchgParam.T_StationCommon.T_Input_Quality_HoleNumber.diInput1 > T_NovRam.T_Parameter.T_PartAnalysis[gciStationSt1].adiNumberHole[ciMaxWP]) THEN
			T_ExchgParam.T_StationCommon.T_Input_Quality_HoleNumber.diInput1:=T_NovRam.T_Parameter.T_PartAnalysis[gciStationSt1].adiNumberHole[ciMaxWP];
		END_IF;
	END_IF;

	IF (T_ExchgParam.T_StationCommon.T_Input_Quality_HoleNumber.diInput1 = 0) THEN
		T_ExchgParam.T_StationCommon.T_Input_Quality_HoleNumber.diInput1:=1;
	END_IF;
	T_ExchgParam.T_StationCommon.T_Input_Quality_HoleNumber.xChangeColour:=FALSE;
	T_ExchgParam.T_StationCommon.T_Input_Quality_HoleNumber.xDisable:=FALSE;
	T_ExchgParam.T_StationCommon.T_Button_Quality_Backward.xDisable:=FALSE;
	T_ExchgParam.T_StationCommon.T_Button_Quality_Forward.xDisable:=FALSE;

	T_ExchgParam.T_StationCommon.T_Input_Quality_HoleNumber.diInputMin:=T_NovRam.T_Parameter.T_PartAnalysis[gciStationSt1].adiNumberHole[1];
	T_ExchgParam.T_StationCommon.T_Input_Quality_HoleNumber.diInputMax:=T_NovRam.T_Parameter.T_PartAnalysis[gciStationSt1].adiNumberHole[ciMaxWP];

	IF (T_ExchgParam.T_StationCommon.T_Input_Quality_HoleNumber.diInput1 < T_ExchgParam.T_StationCommon.T_Input_Quality_HoleNumber.diInputMin) THEN
		T_ExchgParam.T_StationCommon.T_Input_Quality_HoleNumber.diInput1:=T_ExchgParam.T_StationCommon.T_Input_Quality_HoleNumber.diInputMin;
	END_IF;
	IF (T_ExchgParam.T_StationCommon.T_Input_Quality_HoleNumber.diInput1 > T_ExchgParam.T_StationCommon.T_Input_Quality_HoleNumber.diInputMax) THEN
		T_ExchgParam.T_StationCommon.T_Input_Quality_HoleNumber.diInput1:=T_ExchgParam.T_StationCommon.T_Input_Quality_HoleNumber.diInputMax;
	END_IF;

	FBWrapWPQuality(	diHoleNumber:= T_ExchgParam.T_StationCommon.T_Input_Quality_HoleNumber.diInput1,
						T_PartAnalysis:= T_NovRAM.T_Parameter.T_PartAnalysis[gciStationSt1]);

(* Ausgabe der Parameter für die Part Analysis *)
	T_ExchgParam.T_PartQuality.bPartQualityStation:=FBWrapWPQuality.T_DataOut.bHole_WorkPartQuality;
	T_ExchgParam.T_PartQuality.rActualFirstHCPositionStation:=FBWrapWPQuality.T_DataOut.rHole_FirstHC;
	T_ExchgParam.T_PartQuality.iHCCounterStation:=FBWrapWPQuality.T_DataOut.iHole_HCCounter;
	T_ExchgParam.T_PartQuality.iHCCounterCenteringStation:=FBWrapWPQuality.T_DataOut.iHole_HCCounterCentering;
	T_ExchgParam.T_PartQuality.iHCCounterTorqueStation:=FBWrapWPQuality.T_DataOut.iHole_HCCounterTorque;
	T_ExchgParam.T_PartQuality.iHCCounterSpeedStation:=FBWrapWPQuality.T_DataOut.iHole_HCCounterSpeed;
	T_ExchgParam.T_PartQuality.tCycleTimeStation:=DINT_TO_TIME(FBWrapWPQuality.T_DataOut.diHole_CycleTime);
	T_ExchgParam.T_PartQuality.tWorkTimeStation:=DINT_TO_TIME(FBWrapWPQuality.T_DataOut.diHole_WorkTime);
	T_ExchgParam.T_PartQuality.bInfeedCounterZ:=FBWrapWPQuality.T_DataOut.bHole_InfeedCounterZ;
END_IF;
END_ACTION
ACTION CheckSecurityDeactivate:
IF xActivateLayer4_St1St2 THEN
	xActivateLayer4_St1St2:=FALSE;
	TProcess.T_Ctrle.xEnable:=TRUE;
END_IF;

FailingEdge_PowerSupply_NormalOperate_St1St2(CLK:=gT_SafetyStatus.xEnergyONNormalMode AND NOT(xSecurityKey));
IF FailingEdge_PowerSupply_NormalOperate_St1St2.Q THEN
	gxWP_Analyse_ActiveWork:=FALSE;
	gxWP_Analyse_ActiveInfeed:=FALSE;
	gxWP_Analyse_ActiveCentering:=FALSE;
	IF (NOT(TProcess.T_Ctrle.xDone) AND NOT(TProcess.T_Ctrle.xError)) OR NOT(T_Visu.T_CtrleProcess.xDone) THEN
		TProcess.T_Ctrle.xEnable:=FALSE;
		T_Visu.T_CtrleProcess.xReset:=TRUE;
		RisingEdgeReseTProcess(CLK:=FALSE);
		T_Visu.T_CtrleAction.xDeleteVisuFunction:=TRUE;
		T_StartUp.T_Ctrle.xDeleteAllMessageOverlay:=TRUE;
		T_Visu.T_CtrleAction.xFunctionActive:=FALSE;
		T_StartUp.T_State.xBlockChangeMovementVisu:=FALSE;
		xActivateLayer4_St1St2:=TRUE;
		xDeleteProcessFlag_St1St2:=TRUE;
		xActivateMessage:=TRUE;
		IF NOT(TProcess.T_Ctrle.xDone) AND NOT(TProcess.T_Ctrle.xError) AND T_StartUp.T_State.xCompleted THEN
			xProcessEnded:=TRUE;
		END_IF;
	ELSE
		xActivateMessage:=TRUE;
	END_IF;
END_IF;

FailingEdge_PowerSupply_SetupOperateA(CLK:=	(gT_SafetyStatus.xEnergyONSetupModeASt1) AND xSecurityKey AND (iSetupMode = 1));
IF FailingEdge_PowerSupply_SetupOperateA.Q THEN
	gxWP_Analyse_ActiveWork:=FALSE;
	gxWP_Analyse_ActiveInfeed:=FALSE;
	gxWP_Analyse_ActiveCentering:=FALSE;
	IF ((NOT(TProcess.T_Ctrle.xDone) AND NOT(TProcess.T_Ctrle.xError)) OR NOT(T_Visu.T_CtrleProcess.xDone)) THEN
		IF NOT(T_ExchgParam.T_SafetyCtrl.xSetupOperateA_EnergyON) THEN
			TProcess.T_Ctrle.xEnable:=FALSE;
			T_Visu.T_CtrleProcess.xReset:=TRUE;
			RisingEdgeReseTProcess(CLK:=FALSE);
			T_Visu.T_CtrleAction.xDeleteVisuFunction:=TRUE;
			T_StartUp.T_Ctrle.xDeleteAllMessageOverlay:=TRUE;
			T_Visu.T_CtrleAction.xFunctionActive:=FALSE;
			T_StartUp.T_State.xBlockChangeMovementVisu:=FALSE;
			xActivateLayer4_St1St2:=TRUE;
			xDeleteProcessFlag_St1St2:=TRUE;
		END_IF;
		xActivateMessage:=TRUE;
	ELSE
		xActivateMessage:=TRUE;
	END_IF;
END_IF;

FailingEdge_PowerSupply_SetupOperateB(CLK:=	(gT_SafetyStatus.xEnergyONSetupModeBSt1) AND xSecurityKey AND (iSetupMode = 2));
IF FailingEdge_PowerSupply_SetupOperateB.Q THEN
	gxWP_Analyse_ActiveWork:=FALSE;
	gxWP_Analyse_ActiveInfeed:=FALSE;
	gxWP_Analyse_ActiveCentering:=FALSE;
	T_Visu.T_CtrleAction.xDeleteVisuFunction:=TRUE;
	T_StartUp.T_Ctrle.xDeleteAllMessageOverlay:=TRUE;
	T_Visu.T_CtrleAction.xFunctionActive:=FALSE;
	T_StartUp.T_State.xBlockChangeMovementVisu:=FALSE;
	xActivateMessage:=TRUE;
END_IF;

IF xActivateMessage AND T_StartUp.T_State.xCompleted THEN
	TONForceMessage(IN:=TRUE,PT:=T#1s);
	IF (T_ExchgParam.T_Visu.T_Message.iState <> 228) AND (T_ExchgParam.T_Visu.T_Message.iState <> 401) AND
	     NOT((T_ExchgParam.T_Visu.T_Message.iState >= 310) AND (T_ExchgParam.T_Visu.T_Message.iState <= 314)) THEN
		T_ExchgParam.T_Visu.T_Message.iState:=279;	(* Warnung: Sicherheitskreis angesprochen ! *)
	END_IF;
	IF TONForceMessage.Q THEN
		IF NOT(gT_SafetyStatus.xEnergyONNormalMode) THEN
			T_ExchgParam.T_SafetyCtrl.xOpenSecurityDoorMachine:=TRUE;
		END_IF;
		TONForceMessage(IN:=FALSE);
		xActivateMessage:=FALSE;
	END_IF;
ELSE
	TONForceMessage(IN:=FALSE);
	xActivateMessage:=FALSE;
END_IF;

